KUKA KRL program: MyProgram_290().src

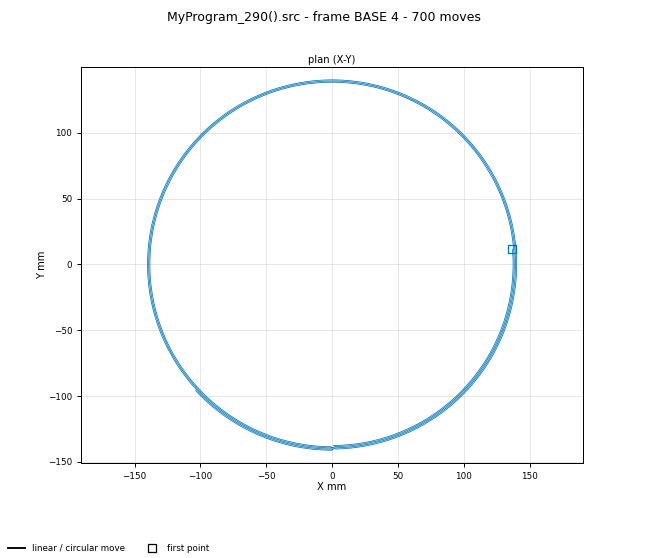
[picture p0: tool path of MyProgram_290().src in frame BASE 4, 700 of 700 moves have a stored position in this frame; points joined in program order, loops and branches not executed]
&ACCESS RVP
&REL 1
&PARAM TEMPLATE = C:\KRC\Roboter\Template\vorgabe
&PARAM EDITMASK = *
DEF MyProgram_290()
; ---- Setting reference (Base) ----
$BASE = BASE_DATA[4]

; --------------------------
; ---- Setting tool (TCP) ----
$TOOL = TOOL_DATA[3]
; --------------------------

$VEL.CP = VEL_APROX_PRINT
Startdeposition()
$VEL.CP = VEL_PRINT
LIN {X 136.961,Y 11.6597,Z 176,A 6.5071,B 7.0853,C 0.2456,E1 7.2488,E2 445.5643} C_DIS
LIN {X 137.2072,Y 8.2752,Z 176,A 5.0839,B 7.0851,C 0.2498,E1 7.2491,E2 446.9898} C_DIS
LIN {X 137.3693,Y 4.9131,Z 176,A 3.7512,B 7.0851,C 0.2525,E1 7.2492,E2 448.3148} C_DIS
LIN {X 137.4448,Y 1.8462,Z 176,A 2.5387,B 7.0849,C 0.2549,E1 7.2493,E2 449.52} C_DIS
LIN {X 137.4365,Y -2.3473,Z 176,A 0.7551,B 7.0847,C 0.2606,E1 7.2493,E2 451.3095} C_DIS
LIN {X 137.322,Y -6.1279,Z 176,A -0.7415,B 7.0847,C 0.2637,E1 7.2491,E2 452.7974} C_DIS
LIN {X 137.1485,Y -9.2287,Z 176,A -2.0117,B 7.0845,C 0.2669,E1 7.2489,E2 454.0657} C_DIS
LIN {X 136.9306,Y -12.0198,Z 176,A -3.1786,B 7.0844,C 0.2703,E1 7.2486,E2 455.2336} C_DIS
LIN {X 136.5827,Y -15.4933,Z 176,A -4.5856,B 7.0843,C 0.2736,E1 7.2482,E2 456.6358} C_DIS
LIN {X 136.1872,Y -18.6525,Z 176,A -5.8882,B 7.0841,C 0.2769,E1 7.2477,E2 457.9365} C_DIS
LIN {X 135.7668,Y -21.4897,Z 176,A -7.0624,B 7.0841,C 0.2799,E1 7.2473,E2 459.1091} C_DIS
LIN {X 135.2243,Y -24.6745,Z 176,A -8.4059,B 7.0839,C 0.2837,E1 7.2466,E2 460.4533} C_DIS
LIN {X 134.6158,Y -27.8022,Z 176,A -9.6822,B 7.0837,C 0.2865,E1 7.2459,E2 461.7243} C_DIS
LIN {X 133.8994,Y -31.0705,Z 176,A -11.0574,B 7.0837,C 0.29,E1 7.2451,E2 463.0983} C_DIS
LIN {X 133.1148,Y -34.2762,Z 176,A -12.4299,B 7.0834,C 0.2938,E1 7.2441,E2 464.4717} C_DIS
LIN {X 132.1526,Y -37.8229,Z 176,A -13.9111,B 7.0834,C 0.2972,E1 7.243,E2 465.948} C_DIS
LIN {X 131.3555,Y -40.4966,Z 176,A -15.0746,B 7.0832,C 0.3004,E1 7.2421,E2 467.1125} C_DIS
LIN {X 130.2621,Y -43.8883,Z 176,A -16.5343,B 7.083,C 0.304,E1 7.2408,E2 468.5704} C_DIS
LIN {X 129.0209,Y -47.4183,Z 176,A -18.0428,B 7.0829,C 0.3073,E1 7.2394,E2 470.074} C_DIS
LIN {X 127.9868,Y -50.1363,Z 176,A -19.2347,B 7.0828,C 0.3102,E1 7.2382,E2 471.2643} C_DIS
LIN {X 126.5088,Y -53.7624,Z 176,A -20.8363,B 7.0826,C 0.3141,E1 7.2365,E2 472.8637} C_DIS
LIN {X 125.2738,Y -56.576,Z 176,A -22.1179,B 7.0824,C 0.3175,E1 7.235,E2 474.1465} C_DIS
LIN {X 123.656,Y -60.0339,Z 176,A -23.6578,B 7.0823,C 0.3207,E1 7.2332,E2 475.6815} C_DIS
LIN {X 122.2692,Y -62.8062,Z 176,A -24.9451,B 7.0821,C 0.324,E1 7.2315,E2 476.9694} C_DIS
LIN {X 120.3748,Y -66.3676,Z 176,A -26.6709,B 7.0819,C 0.3291,E1 7.2292,E2 478.7026} C_DIS
LIN {X 118.274,Y -70.0435,Z 176,A -28.4372,B 7.0817,C 0.3336,E1 7.2268,E2 480.4708} C_DIS
LIN {X 116.0055,Y -73.7401,Z 176,A -30.1691,B 7.0815,C 0.3367,E1 7.2242,E2 482.1948} C_DIS
LIN {X 113.6894,Y -77.2622,Z 176,A -31.8872,B 7.0814,C 0.3403,E1 7.2215,E2 483.9095} C_DIS
LIN {X 111.1496,Y -80.8734,Z 176,A -33.6975,B 7.0812,C 0.3441,E1 7.2186,E2 485.7178} C_DIS
LIN {X 108.4882,Y -84.41,Z 176,A -35.4665,B 7.0811,C 0.3471,E1 7.2156,E2 487.4788} C_DIS
LIN {X 106.0889,Y -87.4067,Z 176,A -37.1314,B 7.0808,C 0.3519,E1 7.2127,E2 489.1535} C_DIS
LIN {X 103.154,Y -90.8515,Z 176,A -38.9691,B 7.0806,C 0.3553,E1 7.2093,E2 490.9868} C_DIS
LIN {X 100.4201,Y -93.8646,Z 176,A -40.5682,B 7.0806,C 0.3572,E1 7.2063,E2 492.5751} C_DIS
LIN {X 97.5463,Y -96.8473,Z 176,A -42.3208,B 7.0803,C 0.3613,E1 7.2029,E2 494.3327} C_DIS
LIN {X 94.6495,Y -99.6812,Z 176,A -43.9576,B 7.0803,C 0.3639,E1 7.1996,E2 495.9643} C_DIS
LIN {X 91.5167,Y -102.5643,Z 176,A -45.7287,B 7.08,C 0.3674,E1 7.1959,E2 497.7366} C_DIS
LIN {X 88.1549,Y -105.4678,Z 176,A -47.5543,B 7.0799,C 0.3705,E1 7.1921,E2 499.5605} C_DIS
LIN {X 84.7062,Y -108.2571,Z 176,A -49.3096,B 7.0798,C 0.3723,E1 7.1883,E2 501.3055} C_DIS
LIN {X 81.738,Y -110.5159,Z 176,A -50.8436,B 7.0796,C 0.3748,E1 7.1848,E2 502.8383} C_DIS
LIN {X 78.8688,Y -112.5814,Z 176,A -52.4099,B 7.0794,C 0.379,E1 7.1812,E2 504.4177} C_DIS
LIN {X 75.2187,Y -115.0523,Z 176,A -54.1125,B 7.0794,C 0.3797,E1 7.1773,E2 506.1046} C_DIS
LIN {X 71.7738,Y -117.2315,Z 176,A -55.8334,B 7.0792,C 0.3828,E1 7.1732,E2 507.8297} C_DIS
LIN {X 68.4893,Y -119.1809,Z 176,A -57.3647,B 7.0792,C 0.3843,E1 7.1695,E2 509.3546} C_DIS
LIN {X 65.2782,Y -120.969,Z 176,A -58.9833,B 7.0789,C 0.388,E1 7.1656,E2 510.9855} C_DIS
LIN {X 61.5873,Y -122.8897,Z 176,A -60.5947,B 7.0789,C 0.3883,E1 7.1616,E2 512.5826} C_DIS
LIN {X 58.8048,Y -124.2432,Z 176,A -61.8707,B 7.0789,C 0.3898,E1 7.1584,E2 513.8578} C_DIS
LIN {X 55.3382,Y -125.8275,Z 176,A -63.4438,B 7.0787,C 0.3916,E1 7.1544,E2 515.4301} C_DIS
LIN {X 52.6854,Y -126.9586,Z 176,A -64.6529,B 7.0787,C 0.3932,E1 7.1512,E2 516.641} C_DIS
LIN {X 49.0097,Y -128.4248,Z 176,A -66.2681,B 7.0786,C 0.3945,E1 7.1471,E2 518.2531} C_DIS
LIN {X 46.1618,Y -129.4738,Z 176,A -67.5214,B 7.0786,C 0.3957,E1 7.1438,E2 519.5057} C_DIS
LIN {X 42.9006,Y -130.591,Z 176,A -68.9539,B 7.0784,C 0.3971,E1 7.14,E2 520.9387} C_DIS
LIN {X 39.5175,Y -131.6552,Z 176,A -70.406,B 7.0784,C 0.3981,E1 7.1361,E2 522.3886} C_DIS
LIN {X 36.5593,Y -132.5059,Z 176,A -71.6852,B 7.0784,C 0.3991,E1 7.1327,E2 523.668} C_DIS
LIN {X 33.0127,Y -133.4355,Z 176,A -73.2026,B 7.0783,C 0.4002,E1 7.1286,E2 525.1851} C_DIS
LIN {X 30.3656,Y -134.0604,Z 176,A -74.339,B 7.0783,C 0.4011,E1 7.1255,E2 526.3226} C_DIS
LIN {X 26.6091,Y -134.8586,Z 176,A -75.9189,B 7.0782,C 0.4019,E1 7.1211,E2 527.9009} C_DIS
LIN {X 23.418,Y -135.4491,Z 176,A -77.2633,B 7.0782,C 0.4026,E1 7.1174,E2 529.245} C_DIS
LIN {X 20.2378,Y -135.9607,Z 176,A -78.5988,B 7.0781,C 0.4033,E1 7.1138,E2 530.5804} C_DIS
LIN {X 17.4061,Y -136.3506,Z 176,A -79.765,B 7.0781,C 0.4034,E1 7.1105,E2 531.744} C_DIS
LIN {X 14.2534,Y -136.7161,Z 176,A -81.0999,B 7.0781,C 0.4042,E1 7.1068,E2 533.0813} C_DIS
LIN {X 10.7874,Y -137.0347,Z 176,A -82.5446,B 7.0781,C 0.4046,E1 7.1028,E2 534.526} C_DIS
LIN {X 8.1562,Y -137.2145,Z 176,A -83.6805,B 7.078,C 0.4055,E1 7.0996,E2 535.6671} C_DIS
LIN {X 4.9131,Y -137.3693,Z 176,A -85.0082,B 7.078,C 0.4055,E1 7.0959,E2 536.9922} C_DIS
LIN {X 1.0091,Y -137.4517,Z 176,A -86.2503,B 7.0783,C 0.3996,E1 7.0926,E2 538.1854} C_DIS
Enddeposition()
LIN {X 1.0091,Y -137.4517,Z 176,A -86.2503,B 7.0783,C 0.3996,E1 7.0926,E2 538.1854} C_DIS
Startdeposition()
$VEL.CP = VEL_PRINT
LIN {X 2.5254,Y -138.3393,Z 176,A -85.3198,B 7.0556,C 0.3987,E1 7.0725,E2 537.2546} C_DIS
LIN {X 6.9228,Y -138.1889,Z 176,A -83.5465,B 7.0556,C 0.399,E1 7.0774,E2 535.4868} C_DIS
LIN {X 10.7421,Y -137.9461,Z 176,A -81.9791,B 7.0556,C 0.3988,E1 7.0818,E2 533.9208} C_DIS
LIN {X 13.4601,Y -137.706,Z 176,A -80.8485,B 7.0556,C 0.3984,E1 7.0849,E2 532.7896} C_DIS
LIN {X 17.2708,Y -137.2818,Z 176,A -78.452,B 7.0564,C 0.3842,E1 7.0919,E2 530.2856} C_DIS
LIN {X 23.2033,Y -136.4032,Z 176,A -76.7282,B 7.0558,C 0.3955,E1 7.0963,E2 528.6605} C_DIS
LIN {X 27.2216,Y -135.6582,Z 176,A -75.0014,B 7.0558,C 0.3938,E1 7.1011,E2 526.9282} C_DIS
LIN {X 30.8555,Y -134.8775,Z 176,A -73.2676,B 7.0561,C 0.3893,E1 7.1059,E2 525.1678} C_DIS
LIN {X 34.0474,Y -134.1073,Z 176,A -72.1782,B 7.0559,C 0.3928,E1 7.1087,E2 524.113} C_DIS
LIN {X 37.8887,Y -133.0746,Z 176,A -70.5771,B 7.0559,C 0.3921,E1 7.113,E2 522.5169} C_DIS
LIN {X 40.8202,Y -132.2037,Z 176,A -69.3143,B 7.056,C 0.391,E1 7.1164,E2 521.2536} C_DIS
LIN {X 44.7183,Y -130.9376,Z 176,A -67.5846,B 7.0561,C 0.3887,E1 7.121,E2 519.5184} C_DIS
LIN {X 48.2676,Y -129.6699,Z 176,A -66.1821,B 7.0561,C 0.3897,E1 7.1246,E2 518.1355} C_DIS
LIN {X 51.4027,Y -128.4595,Z 176,A -64.8772,B 7.0561,C 0.3897,E1 7.128,E2 516.8409} C_DIS
LIN {X 54.2024,Y -127.3051,Z 176,A -63.4709,B 7.0563,C 0.3855,E1 7.1317,E2 515.4138} C_DIS
LIN {X 56.8151,Y -126.1591,Z 176,A -62.182,B 7.0565,C 0.3821,E1 7.135,E2 514.1098} C_DIS
LIN {X 60.1001,Y -124.6281,Z 176,A -60.6977,B 7.0566,C 0.3804,E1 7.1387,E2 512.6265} C_DIS
LIN {X 63.3527,Y -123.0073,Z 176,A -59.1577,B 7.0567,C 0.3776,E1 7.1426,E2 511.0807} C_DIS
LIN {X 67.4632,Y -120.803,Z 176,A -57.3038,B 7.0568,C 0.3762,E1 7.1471,E2 509.2355} C_DIS
LIN {X 72.6683,Y -117.7453,Z 176,A -54.8126,B 7.057,C 0.3724,E1 7.1531,E2 506.7434} C_DIS
LIN {X 76.3854,Y -115.3685,Z 176,A -53.0068,B 7.0572,C 0.3697,E1 7.1573,E2 504.9387} C_DIS
LIN {X 81.0498,Y -112.1403,Z 176,A -49.8357,B 7.0581,C 0.3507,E1 7.1648,E2 501.6571} C_DIS
LIN {X 86.6426,Y -107.8779,Z 176,A -47.9887,B 7.0574,C 0.3647,E1 7.1685,E2 499.948} C_DIS
LIN {X 92.5705,Y -102.8361,Z 176,A -44.8865,B 7.0576,C 0.3606,E1 7.1751,E2 496.8588} C_DIS
LIN {X 96.6443,Y -99.0176,Z 176,A -42.3516,B 7.0581,C 0.3518,E1 7.1803,E2 494.2927} C_DIS
LIN {X 102.4902,Y -92.953,Z 176,A -39.1952,B 7.0581,C 0.3504,E1 7.1863,E2 491.1765} C_DIS
LIN {X 106.6921,Y -88.0984,Z 176,A -36.5612,B 7.0584,C 0.3449,E1 7.1911,E2 488.5434} C_DIS
LIN {X 109.9326,Y -84.0198,Z 176,A -34.3714,B 7.0587,C 0.3393,E1 7.1949,E2 486.3473} C_DIS
LIN {X 111.7517,Y -81.5857,Z 176,A -33.0115,B 7.0589,C 0.3345,E1 7.1971,E2 484.9731} C_DIS
LIN {X 114.075,Y -78.3031,Z 176,A -31.3295,B 7.0591,C 0.3301,E1 7.1998,E2 483.2873} C_DIS
LIN {X 116.3731,Y -74.8457,Z 176,A -29.6118,B 7.0593,C 0.3259,E1 7.2024,E2 481.5681} C_DIS
LIN {X 118.7096,Y -71.0817,Z 176,A -27.9699,B 7.0593,C 0.3249,E1 7.2048,E2 479.9496} C_DIS
LIN {X 120.5701,Y -67.8775,Z 176,A -26.3198,B 7.0596,C 0.3189,E1 7.2071,E2 478.2829} C_DIS
LIN {X 122.7224,Y -63.9013,Z 176,A -24.5849,B 7.0597,C 0.3166,E1 7.2094,E2 476.564} C_DIS
LIN {X 124.4953,Y -60.3781,Z 176,A -22.1195,B 7.0606,C 0.2966,E1 7.2125,E2 473.9882} C_DIS
LIN {X 127.1523,Y -54.5563,Z 176,A -20.3094,B 7.0602,C 0.3055,E1 7.2144,E2 472.2855} C_DIS
LIN {X 129.6051,Y -48.4406,Z 176,A -17.6421,B 7.0605,C 0.2993,E1 7.2171,E2 469.6237} C_DIS
LIN {X 130.7909,Y -45.1415,Z 176,A -16.2657,B 7.0605,C 0.2967,E1 7.2184,E2 468.2557} C_DIS
LIN {X 131.9779,Y -41.5469,Z 176,A -14.7467,B 7.0607,C 0.2933,E1 7.2197,E2 466.7415} C_DIS
LIN {X 133.0729,Y -37.8948,Z 176,A -13.2187,B 7.0609,C 0.2899,E1 7.2209,E2 465.2187} C_DIS
LIN {X 134.2589,Y -33.4503,Z 176,A -11.3485,B 7.0611,C 0.2852,E1 7.2222,E2 463.3511} C_DIS
LIN {X 135.0961,Y -29.8924,Z 176,A -9.8374,B 7.0612,C 0.281,E1 7.2231,E2 461.8389} C_DIS
LIN {X 136.0368,Y -25.2694,Z 176,A -7.6229,B 7.0616,C 0.2705,E1 7.2243,E2 459.5889} C_DIS
LIN {X 136.6167,Y -21.9198,Z 176,A -6.5809,B 7.0616,C 0.2734,E1 7.2248,E2 458.5929} C_DIS
LIN {X 136.9695,Y -19.5809,Z 176,A -5.5854,B 7.0616,C 0.2703,E1 7.2252,E2 457.5944} C_DIS
LIN {X 137.3908,Y -16.3656,Z 176,A -4.2291,B 7.0618,C 0.2662,E1 7.2256,E2 456.2352} C_DIS
LIN {X 138.1174,Y -8.2298,Z 176,A -1.086,B 7.062,C 0.2611,E1 7.2264,E2 453.1201} C_DIS
LIN {X 138.2614,Y -5.2795,Z 176,A 0.2729,B 7.0622,C 0.255,E1 7.2265,E2 451.7427} C_DIS
LIN {X 138.3608,Y -0.7908,Z 176,A 2.1226,B 7.0624,C 0.2498,E1 7.2265,E2 449.8927} C_DIS
LIN {X 138.3336,Y 2.8695,Z 176,A 3.5024,B 7.0624,C 0.2481,E1 7.2265,E2 448.5292} C_DIS
LIN {X 138.2205,Y 6.2935,Z 176,A 5.1475,B 7.0627,C 0.2397,E1 7.2264,E2 446.8537} C_DIS
LIN {X 137.9761,Y 10.3308,Z 176,A 6.6024,B 7.0627,C 0.2391,E1 7.2261,E2 445.4258} C_DIS
LIN {X 137.1498,Y 18.2779,Z 176,A 9.844,B 7.063,C 0.2309,E1 7.2251,E2 442.1904} C_DIS
LIN {X 136.704,Y 21.3562,Z 176,A 11.0883,B 7.0631,C 0.2281,E1 7.2246,E2 440.9507} C_DIS
LIN {X 136.1551,Y 24.6144,Z 176,A 12.4408,B 7.0632,C 0.2245,E1 7.2239,E2 439.5991} C_DIS
LIN {X 135.0836,Y 29.9503,Z 176,A 14.6215,B 7.0634,C 0.2196,E1 7.2227,E2 437.4263} C_DIS
LIN {X 134.4438,Y 32.6949,Z 176,A 15.8649,B 7.0635,C 0.2149,E1 7.2219,E2 436.1722} C_DIS
LIN {X 133.332,Y 36.9684,Z 176,A 17.6054,B 7.0636,C 0.2115,E1 7.2206,E2 434.4417} C_DIS
LIN {X 132.3059,Y 40.4861,Z 176,A 19.0601,B 7.0637,C 0.2085,E1 7.2194,E2 432.994} C_DIS
LIN {X 131.194,Y 43.9563,Z 176,A 20.5614,B 7.0638,C 0.2045,E1 7.2181,E2 431.4927} C_DIS
LIN {X 130.0878,Y 47.1295,Z 176,A 21.9276,B 7.0639,C 0.2012,E1 7.2169,E2 430.1288} C_DIS
LIN {X 128.7264,Y 50.7334,Z 176,A 23.7502,B 7.0642,C 0.1928,E1 7.215,E2 428.2762} C_DIS
LIN {X 126.8213,Y 55.322,Z 176,A 25.4906,B 7.0642,C 0.1932,E1 7.2131,E2 426.575} C_DIS
LIN {X 125.3764,Y 58.5231,Z 176,A 27.0649,B 7.0643,C 0.1872,E1 7.2113,E2 424.9847} C_DIS
LIN {X 123.8041,Y 61.7808,Z 176,A 28.3809,B 7.0643,C 0.1868,E1 7.2097,E2 423.691} C_DIS
LIN {X 122.2976,Y 64.7103,Z 176,A 29.765,B 7.0644,C 0.1829,E1 7.2079,E2 422.3036} C_DIS
LIN {X 116.9096,Y 74.0045,Z 176,A 34.0572,B 7.0646,C 0.1749,E1 7.2019,E2 418.0296} C_DIS
LIN {X 114.3482,Y 77.9047,Z 176,A 36.1172,B 7.0648,C 0.168,E1 7.1986,E2 415.9526} C_DIS
LIN {X 111.806,Y 81.5111,Z 176,A 37.9057,B 7.0648,C 0.1644,E1 7.1957,E2 414.1682} C_DIS
LIN {X 108.7844,Y 85.5012,Z 176,A 39.7845,B 7.0649,C 0.1632,E1 7.1925,E2 412.3131} C_DIS
LIN {X 106.3447,Y 88.5179,Z 176,A 41.4898,B 7.065,C 0.1579,E1 7.1895,E2 410.5948} C_DIS
LIN {X 103.8728,Y 91.4058,Z 176,A 43.0987,B 7.0651,C 0.1539,E1 7.1865,E2 408.981} C_DIS
LIN {X 100.77,Y 94.8152,Z 176,A 44.9608,B 7.0651,C 0.1507,E1 7.183,E2 407.1242} C_DIS
LIN {X 97.5573,Y 98.1176,Z 176,A 46.9196,B 7.0653,C 0.1459,E1 7.1791,E2 405.1584} C_DIS
LIN {X 94.2943,Y 101.2575,Z 176,A 48.4305,B 7.0653,C 0.1487,E1 7.1762,E2 403.693} C_DIS
LIN {X 92.1308,Y 103.2301,Z 176,A 49.8679,B 7.0653,C 0.1424,E1 7.1731,E2 402.227} C_DIS
LIN {X 88.6833,Y 106.2068,Z 176,A 51.7248,B 7.0654,C 0.1394,E1 7.1692,E2 400.3735} C_DIS
LIN {X 85.3526,Y 108.901,Z 176,A 53.4781,B 7.0654,C 0.1366,E1 7.1654,E2 398.6224} C_DIS
LIN {X 81.7479,Y 111.6325,Z 176,A 55.3312,B 7.0655,C 0.1337,E1 7.1612,E2 396.7716} C_DIS
LIN {X 74.1764,Y 116.8011,Z 176,A 59.2347,B 7.0657,C 0.1259,E1 7.1521,E2 392.8545} C_DIS
LIN {X 69.8268,Y 119.4521,Z 176,A 61.1523,B 7.0657,C 0.1261,E1 7.1476,E2 390.9609} C_DIS
LIN {X 65.895,Y 121.6656,Z 176,A 63.0289,B 7.0657,C 0.1233,E1 7.143,E2 389.0833} C_DIS
LIN {X 60.1682,Y 124.5956,Z 176,A 65.4693,B 7.0657,C 0.1237,E1 7.137,E2 386.6709} C_DIS
LIN {X 56.1062,Y 126.4762,Z 176,A 67.4503,B 7.0657,C 0.1193,E1 7.1319,E2 384.6741} C_DIS
LIN {X 51.4384,Y 128.4451,Z 176,A 69.4867,B 7.0658,C 0.118,E1 7.1267,E2 382.6455} C_DIS
LIN {X 48.0789,Y 129.7406,Z 176,A 70.9544,B 7.0658,C 0.1169,E1 7.1228,E2 381.181} C_DIS
LIN {X 45.1935,Y 130.7729,Z 176,A 72.2552,B 7.0658,C 0.1152,E1 7.1194,E2 379.8765} C_DIS
LIN {X 41.978,Y 131.8402,Z 176,A 73.6416,B 7.0658,C 0.1142,E1 7.1157,E2 378.4923} C_DIS
LIN {X 38.3573,Y 132.9398,Z 176,A 75.1467,B 7.0658,C 0.1139,E1 7.1117,E2 376.9953} C_DIS
LIN {X 34.814,Y 133.9128,Z 176,A 76.8878,B 7.066,C 0.1092,E1 7.1069,E2 375.2271} C_DIS
LIN {X 31.0115,Y 134.8419,Z 176,A 78.3311,B 7.066,C 0.111,E1 7.1031,E2 373.8064} C_DIS
LIN {X 25.4929,Y 135.9941,Z 176,A 80.5918,B 7.066,C 0.1109,E1 7.0969,E2 371.5556} C_DIS
LIN {X 22.3228,Y 136.5501,Z 176,A 82.0724,B 7.066,C 0.1078,E1 7.0928,E2 370.0569} C_DIS
LIN {X 17.0323,Y 137.3112,Z 176,A 84.0919,B 7.066,C 0.1101,E1 7.0873,E2 368.0624} C_DIS
LIN {X 12.0718,Y 137.8351,Z 176,A 86.0722,B 7.066,C 0.1108,E1 7.0818,E2 366.0935} C_DIS
LIN {X 7.3371,Y 138.168,Z 176,A 88.2612,B 7.066,C 0.1069,E1 7.0756,E2 363.8774} C_DIS
LIN {X 2.8858,Y 138.3333,Z 176,A 90.1438,B 7.066,C 0.1062,E1 7.0704,E2 361.9909} C_DIS
LIN {X -1.2214,Y 138.3576,Z 176,A 91.6876,B 7.066,C 0.1086,E1 7.0661,E2 360.4674} C_DIS
LIN {X -4.5578,Y 138.2889,Z 176,A 93.9422,B 7.0662,C 0.0953,E1 7.0595,E2 358.1041} C_DIS
LIN {X -10.7096,Y 137.9485,Z 176,A 95.5331,B 7.0659,C 0.1104,E1 7.0554,E2 356.6349} C_DIS
LIN {X -18.6513,Y 137.1008,Z 176,A 99.4322,B 7.0661,C 0.1026,E1 7.0444,E2 352.664} C_DIS
LIN {X -22.6044,Y 136.5031,Z 176,A 100.4171,B 7.0659,C 0.1134,E1 7.0419,E2 351.7636} C_DIS
LIN {X -24.5794,Y 136.1614,Z 176,A 101.5762,B 7.0659,C 0.1089,E1 7.0386,E2 350.5642} C_DIS
LIN {X -29.0231,Y 135.2838,Z 176,A 103.4719,B 7.0659,C 0.1097,E1 7.0334,E2 348.6671} C_DIS
LIN {X -32.4353,Y 134.5063,Z 176,A 104.8068,B 7.0659,C 0.1123,E1 7.0298,E2 347.3473} C_DIS
LIN {X -36.4117,Y 133.4871,Z 176,A 106.5159,B 7.0659,C 0.1134,E1 7.0252,E2 345.6383} C_DIS
LIN {X -40.6365,Y 132.2599,Z 176,A 108.3838,B 7.0659,C 0.1142,E1 7.0202,E2 343.7658} C_DIS
LIN {X -44.2376,Y 131.1004,Z 176,A 110.5174,B 7.0659,C 0.1075,E1 7.0144,E2 341.5623} C_DIS
LIN {X -48.7219,Y 129.4997,Z 176,A 111.8393,B 7.0659,C 0.1187,E1 7.0111,E2 340.3231} C_DIS
LIN {X -52.0437,Y 128.2011,Z 176,A 113.3948,B 7.0658,C 0.1192,E1 7.0071,E2 338.759} C_DIS
LIN {X -55.294,Y 126.8333,Z 176,A 114.9898,B 7.0658,C 0.1189,E1 7.0029,E2 337.1483} C_DIS
LIN {X -59.0033,Y 125.1521,Z 176,A 116.8221,B 7.0658,C 0.1189,E1 6.9982,E2 335.2991} C_DIS
LIN {X -63.5602,Y 122.9015,Z 176,A 118.7168,B 7.0658,C 0.1246,E1 6.9936,E2 333.4323} C_DIS
LIN {X -66.6076,Y 121.2769,Z 176,A 120.6249,B 7.0658,C 0.1199,E1 6.9888,E2 331.4655} C_DIS
LIN {X -70.2498,Y 119.2036,Z 176,A 121.6918,B 7.0656,C 0.1317,E1 6.9864,E2 330.4835} C_DIS
LIN {X -74.9128,Y 116.3301,Z 176,A 124.2214,B 7.0656,C 0.1315,E1 6.9803,E2 327.9232} C_DIS
LIN {X -78.1221,Y 114.1993,Z 176,A 125.9356,B 7.0656,C 0.1325,E1 6.9763,E2 326.1956} C_DIS
LIN {X -81.8457,Y 111.5606,Z 176,A 128.0751,B 7.0656,C 0.1323,E1 6.9714,E2 324.0264} C_DIS
LIN {X -84.6797,Y 109.4251,Z 176,A 129.1735,B 7.0654,C 0.1399,E1 6.9691,E2 322.9757} C_DIS
LIN {X -87.6801,Y 107.0361,Z 176,A 130.9221,B 7.0654,C 0.1406,E1 6.9653,E2 321.2085} C_DIS
LIN {X -91.1706,Y 104.0792,Z 176,A 132.9117,B 7.0654,C 0.1429,E1 6.961,E2 319.2086} C_DIS
LIN {X -94.7376,Y 100.8432,Z 176,A 134.7784,B 7.0652,C 0.1484,E1 6.9572,E2 317.3597} C_DIS
LIN {X -97.6555,Y 98.02,Z 176,A 136.5495,B 7.0652,C 0.1507,E1 6.9537,E2 315.5789} C_DIS
LIN {X -100.7775,Y 94.8073,Z 176,A 138.5403,B 7.0652,C 0.1527,E1 6.9498,E2 313.5727} C_DIS
LIN {X -104.0802,Y 91.1694,Z 176,A 140.4595,B 7.065,C 0.1586,E1 6.9463,E2 311.6699} C_DIS
LIN {X -106.5987,Y 88.2111,Z 176,A 142.1398,B 7.065,C 0.1612,E1 6.9433,E2 309.9821} C_DIS
LIN {X -109.2558,Y 84.8981,Z 176,A 143.9146,B 7.0649,C 0.165,E1 6.9402,E2 308.207} C_DIS
LIN {X -111.8062,Y 81.5108,Z 176,A 145.7743,B 7.0649,C 0.1677,E1 6.9371,E2 306.3359} C_DIS
LIN {X -114.4796,Y 77.7107,Z 176,A 147.7115,B 7.0647,C 0.1721,E1 6.934,E2 304.3989} C_DIS
LIN {X -117.2797,Y 73.4173,Z 176,A 149.575,B 7.0645,C 0.1806,E1 6.9312,E2 302.5698} C_DIS
LIN {X -118.8014,Y 70.9276,Z 176,A 151.0457,B 7.0645,C 0.1802,E1 6.9291,E2 301.0675} C_DIS
LIN {X -120.9228,Y 67.2476,Z 176,A 152.8882,B 7.0645,C 0.1836,E1 6.9265,E2 299.2162} C_DIS
LIN {X -122.8738,Y 63.6129,Z 176,A 154.7775,B 7.0644,C 0.1857,E1 6.924,E2 297.3057} C_DIS
LIN {X -125.1706,Y 58.9646,Z 176,A 156.698,B 7.0641,C 0.1941,E1 6.9218,E2 295.4157} C_DIS
LIN {X -126.2768,Y 56.5519,Z 176,A 157.9683,B 7.0641,C 0.1948,E1 6.9203,E2 294.1249} C_DIS
LIN {X -128.3795,Y 51.6012,Z 176,A 160.0918,B 7.0639,C 0.2021,E1 6.918,E2 292.0166} C_DIS
LIN {X -129.8312,Y 47.8368,Z 176,A 161.7888,B 7.0638,C 0.2063,E1 6.9163,E2 290.3179} C_DIS
LIN {X -130.6764,Y 45.4716,Z 176,A 162.8849,B 7.0638,C 0.2084,E1 6.9153,E2 289.2157} C_DIS
LIN {X -131.8419,Y 41.9728,Z 176,A 164.4104,B 7.0636,C 0.2126,E1 6.914,E2 287.6918} C_DIS
LIN {X -132.847,Y 38.6743,Z 176,A 165.8678,B 7.0636,C 0.2162,E1 6.9128,E2 286.232} C_DIS
LIN {X -133.9152,Y 34.8045,Z 176,A 167.552,B 7.0634,C 0.2205,E1 6.9116,E2 284.5467} C_DIS
LIN {X -134.6189,Y 31.9682,Z 176,A 168.7885,B 7.0633,C 0.2236,E1 6.9108,E2 283.3079} C_DIS
LIN {X -135.3494,Y 28.719,Z 176,A 170.5625,B 7.0633,C 0.2225,E1 6.9097,E2 281.4852} C_DIS
LIN {X -136.0605,Y 25.1429,Z 176,A 171.7319,B 7.063,C 0.2311,E1 6.9092,E2 280.3604} C_DIS
LIN {X -136.6305,Y 21.8312,Z 176,A 173.1103,B 7.0629,C 0.2352,E1 6.9085,E2 278.9849} C_DIS
LIN {X -136.9789,Y 19.5148,Z 176,A 174.1998,B 7.0629,C 0.2364,E1 6.9081,E2 277.8811} C_DIS
LIN {X -137.4594,Y 15.79,Z 176,A 175.9795,B 7.0629,C 0.2381,E1 6.9075,E2 276.0744} C_DIS
LIN {X -137.9915,Y 10.1209,Z 176,A 178.1946,B 7.0625,C 0.2466,E1 6.907,E2 273.8794} C_DIS
LIN {X -138.2142,Y 6.4189,Z 176,A 179.6754,B 7.0623,C 0.2517,E1 6.9067,E2 272.4069} C_DIS
LIN {X -138.316,Y 3.584,Z 176,A -179.0267,B 7.0623,C 0.2535,E1 6.9067,E2 271.0944} C_DIS
LIN {X -138.3578,Y -1.247,Z 176,A -176.89,B 7.0621,C 0.2576,E1 6.9067,E2 268.9421} C_DIS
LIN {X -138.2909,Y -4.4889,Z 176,A -175.5269,B 7.062,C 0.2612,E1 6.9067,E2 267.5776} C_DIS
LIN {X -138.0898,Y -8.6788,Z 176,A -173.859,B 7.0618,C 0.267,E1 6.907,E2 265.9199} C_DIS
LIN {X -137.761,Y -12.8878,Z 176,A -172.0353,B 7.0616,C 0.2711,E1 6.9074,E2 264.088} C_DIS
LIN {X -137.3825,Y -16.4352,Z 176,A -170.5282,B 7.0615,C 0.2749,E1 6.9079,E2 262.5782} C_DIS
LIN {X -136.9344,Y -19.8261,Z 176,A -169.1912,B 7.0613,C 0.2799,E1 6.9084,E2 261.2525} C_DIS
LIN {X -136.4284,Y -23.0524,Z 176,A -167.7791,B 7.0612,C 0.283,E1 6.9091,E2 259.8337} C_DIS
LIN {X -135.8712,Y -26.1354,Z 176,A -166.4354,B 7.061,C 0.286,E1 6.9097,E2 258.4851} C_DIS
LIN {X -135.1625,Y -29.5848,Z 176,A -164.9621,B 7.0609,C 0.2899,E1 6.9106,E2 257.011} C_DIS
LIN {X -134.4193,Y -32.7963,Z 176,A -163.5629,B 7.0607,C 0.2933,E1 6.9115,E2 255.6084} C_DIS
LIN {X -133.6143,Y -35.9345,Z 176,A -162.2415,B 7.0606,C 0.2972,E1 6.9124,E2 254.2905} C_DIS
LIN {X -132.61,Y -39.4839,Z 176,A -160.6475,B 7.0604,C 0.3006,E1 6.9137,E2 252.6891} C_DIS
LIN {X -131.703,Y -42.4075,Z 176,A -159.2818,B 7.0604,C 0.3028,E1 6.9149,E2 251.3116} C_DIS
LIN {X -130.0466,Y -47.2436,Z 176,A -157.1409,B 7.0601,C 0.3081,E1 6.9168,E2 249.169} C_DIS
LIN {X -128.3241,Y -51.7385,Z 176,A -155.0842,B 7.0599,C 0.3126,E1 6.9189,E2 247.1055} C_DIS
LIN {X -126.9679,Y -54.9828,Z 176,A -153.6414,B 7.0597,C 0.3166,E1 6.9205,E2 245.6652} C_DIS
LIN {X -125.4556,Y -58.3518,Z 176,A -152.0807,B 7.0596,C 0.3201,E1 6.9223,E2 244.1013} C_DIS
LIN {X -123.8944,Y -61.5978,Z 176,A -150.5429,B 7.0594,C 0.3233,E1 6.9242,E2 242.5585} C_DIS
LIN {X -121.2381,Y -66.6781,Z 176,A -148.2558,B 7.0591,C 0.3304,E1 6.9272,E2 240.2839} C_DIS
LIN {X -119.5646,Y -69.6342,Z 176,A -146.6081,B 7.0591,C 0.3306,E1 6.9295,E2 238.6059} C_DIS
LIN {X -117.2863,Y -73.4067,Z 176,A -144.7695,B 7.0589,C 0.3348,E1 6.9322,E2 236.7664} C_DIS
LIN {X -114.8052,Y -77.2296,Z 176,A -142.8289,B 7.0587,C 0.3385,E1 6.9352,E2 234.8198} C_DIS
LIN {X -112.2223,Y -80.9367,Z 176,A -140.9162,B 7.0585,C 0.3423,E1 6.9383,E2 232.9025} C_DIS
LIN {X -109.4986,Y -84.5849,Z 176,A -139.055,B 7.0583,C 0.3468,E1 6.9415,E2 231.0451} C_DIS
LIN {X -106.7972,Y -87.9714,Z 176,A -137.201,B 7.0582,C 0.3499,E1 6.9447,E2 229.184} C_DIS
LIN {X -103.8757,Y -91.4026,Z 176,A -135.3599,B 7.058,C 0.3541,E1 6.9481,E2 227.3467} C_DIS
LIN {X -101.1595,Y -94.3995,Z 176,A -133.6342,B 7.0578,C 0.3569,E1 6.9514,E2 225.615} C_DIS
LIN {X -98.0463,Y -97.6291,Z 176,A -131.7297,B 7.0577,C 0.3599,E1 6.9551,E2 223.7049} C_DIS
LIN {X -94.9038,Y -100.6864,Z 176,A -129.9244,B 7.0575,C 0.3635,E1 6.9587,E2 221.9014} C_DIS
LIN {X -91.9303,Y -103.4092,Z 176,A -128.1736,B 7.0574,C 0.3655,E1 6.9624,E2 220.1404} C_DIS
LIN {X -88.474,Y -106.3811,Z 176,A -126.2694,B 7.0572,C 0.3686,E1 6.9665,E2 218.2345} C_DIS
LIN {X -84.9058,Y -109.2499,Z 176,A -124.3523,B 7.0571,C 0.3715,E1 6.9707,E2 216.3149} C_DIS
LIN {X -79.3843,Y -113.3261,Z 176,A -121.7445,B 7.0567,C 0.3794,E1 6.9765,E2 213.738} C_DIS
LIN {X -75.2774,Y -116.094,Z 176,A -119.3526,B 7.0567,C 0.3776,E1 6.9822,E2 211.3019} C_DIS
LIN {X -71.1714,Y -118.6561,Z 176,A -117.4373,B 7.0565,C 0.3817,E1 6.9867,E2 209.3983} C_DIS
LIN {X -67.4222,Y -120.826,Z 176,A -115.2033,B 7.0567,C 0.3776,E1 6.9923,E2 207.1068} C_DIS
LIN {X -63.6973,Y -122.8295,Z 176,A -113.9272,B 7.0563,C 0.3867,E1 6.9953,E2 205.8927} C_DIS
LIN {X -60.8532,Y -124.2617,Z 176,A -112.6294,B 7.0562,C 0.3886,E1 6.9985,E2 204.5975} C_DIS
LIN {X -58.1944,Y -125.5284,Z 176,A -111.2678,B 7.0562,C 0.3878,E1 7.002,E2 203.2174} C_DIS
LIN {X -54.5178,Y -127.1689,Z 176,A -109.6743,B 7.056,C 0.3907,E1 7.0061,E2 201.6334} C_DIS
LIN {X -51.3166,Y -128.4942,Z 176,A -108.2341,B 7.056,C 0.392,E1 7.0098,E2 200.1922} C_DIS
LIN {X -48.4312,Y -129.6086,Z 176,A -106.899,B 7.056,C 0.3923,E1 7.0133,E2 198.8499} C_DIS
LIN {X -45.1224,Y -130.7975,Z 176,A -105.4588,B 7.0559,C 0.3938,E1 7.0171,E2 197.4115} C_DIS
LIN {X -41.3185,Y -132.0509,Z 176,A -103.8134,B 7.0558,C 0.3953,E1 7.0215,E2 195.7676} C_DIS
LIN {X -38.1212,Y -133.009,Z 176,A -102.1842,B 7.0559,C 0.3925,E1 7.0259,E2 194.1058} C_DIS
LIN {X -33.4693,Y -134.2541,Z 176,A -100.4503,B 7.0557,C 0.3977,E1 7.0305,E2 192.4054} C_DIS
LIN {X -27.2636,Y -135.6496,Z 176,A -97.8078,B 7.0556,C 0.3989,E1 7.0377,E2 189.7612} C_DIS
LIN {X -20.0589,Y -136.9011,Z 176,A -94.8682,B 7.0554,C 0.4014,E1 7.0458,E2 186.8324} C_DIS
LIN {X -17.1071,Y -137.3023,Z 176,A -93.3739,B 7.0557,C 0.3976,E1 7.05,E2 185.3036} C_DIS
LIN {X -13.139,Y -137.7368,Z 176,A -91.794,B 7.0556,C 0.399,E1 7.0544,E2 183.7325} C_DIS
LIN {X -9.5103,Y -138.036,Z 176,A -90.208,B 7.0556,C 0.3979,E1 7.0588,E2 182.1358} C_DIS
LIN {X -5.4944,Y -138.2531,Z 176,A -88.6422,B 7.0556,C 0.3995,E1 7.0632,E2 180.5822} C_DIS
LIN {X -1.3582,Y -138.3568,Z 176,A -86.8621,B 7.0556,C 0.3983,E1 7.0682,E2 178.7926} C_DIS
LIN {X -1.3582,Y -138.3568,Z 176,A -86.8621,B 7.0556,C 0.3983,E1 7.0682,E2 178.7926} C_DIS
Enddeposition()
LIN {X 1.0282,Y -139.2615,Z 176,A -86.1341,B 7.032,C 0.4064,E1 7.0469,E2 178.1377} C_DIS
Startdeposition()
$VEL.CP = VEL_PRINT
LIN {X -1.8048,Y -139.2572,Z 176,A -87.67,B 7.0317,C 0.4125,E1 7.0425,E2 179.7228} C_DIS
LIN {X -5.3362,Y -139.1656,Z 176,A -89.2451,B 7.0316,C 0.4145,E1 7.038,E2 181.3144} C_DIS
LIN {X -9.8584,Y -138.9187,Z 176,A -91.0825,B 7.0316,C 0.414,E1 7.0329,E2 183.1492} C_DIS
LIN {X -13.4981,Y -138.6122,Z 176,A -92.5369,B 7.0316,C 0.413,E1 7.0289,E2 184.598} C_DIS
LIN {X -17.4777,Y -138.1681,Z 176,A -94.2397,B 7.0316,C 0.4136,E1 7.0241,E2 186.3086} C_DIS
LIN {X -21.1208,Y -137.657,Z 176,A -95.7999,B 7.0316,C 0.4138,E1 7.0198,E2 187.8754} C_DIS
LIN {X -26.5006,Y -136.7235,Z 176,A -97.9446,B 7.0317,C 0.4114,E1 7.014,E2 190.0075} C_DIS
LIN {X -30.016,Y -135.9956,Z 176,A -99.7839,B 7.0315,C 0.4162,E1 7.0088,E2 191.8944} C_DIS
LIN {X -33.5464,Y -135.1689,Z 176,A -100.8984,B 7.0318,C 0.4096,E1 7.0059,E2 192.9603} C_DIS
LIN {X -38.51,Y -133.8389,Z 176,A -103.066,B 7.0318,C 0.4091,E1 7.0001,E2 195.1353} C_DIS
LIN {X -42.0634,Y -132.7637,Z 176,A -104.65,B 7.0318,C 0.4088,E1 6.9958,E2 196.727} C_DIS
LIN {X -45.0781,Y -131.7714,Z 176,A -106.023,B 7.0318,C 0.4088,E1 6.9921,E2 198.109} C_DIS
LIN {X -48.9972,Y -130.3637,Z 176,A -107.698,B 7.032,C 0.4067,E1 6.9878,E2 199.7792} C_DIS
LIN {X -53.2829,Y -128.6721,Z 176,A -109.5801,B 7.0321,C 0.4046,E1 6.9829,E2 201.6598} C_DIS
LIN {X -58.1856,Y -126.5303,Z 176,A -111.784,B 7.0323,C 0.4024,E1 6.9773,E2 203.8643} C_DIS
LIN {X -61.2577,Y -125.0721,Z 176,A -114.2149,B 7.0315,C 0.4156,E1 6.9709,E2 206.4281} C_DIS
LIN {X -67.84,Y -121.63,Z 176,A -116.3911,B 7.0324,C 0.3992,E1 6.9658,E2 208.4915} C_DIS
LIN {X -71.6173,Y -119.4447,Z 176,A -118.184,B 7.0326,C 0.3967,E1 6.9615,E2 210.284} C_DIS
LIN {X -76.3084,Y -116.5033,Z 176,A -120.3041,B 7.0329,C 0.3911,E1 6.9565,E2 212.3835} C_DIS
LIN {X -78.9065,Y -114.7594,Z 176,A -122.3623,B 7.0324,C 0.4,E1 6.9516,E2 214.541} C_DIS
LIN {X -83.312,Y -111.6023,Z 176,A -123.9917,B 7.0331,C 0.388,E1 6.9481,E2 216.0929} C_DIS
LIN {X -86.8271,Y -108.8899,Z 176,A -125.8757,B 7.0331,C 0.3858,E1 6.9439,E2 217.9841} C_DIS
LIN {X -90.3998,Y -105.9428,Z 176,A -127.8118,B 7.0333,C 0.3828,E1 6.9398,E2 219.9237} C_DIS
LIN {X -93.7796,Y -102.9631,Z 176,A -129.6657,B 7.0335,C 0.3794,E1 6.9359,E2 221.7773} C_DIS
LIN {X -96.9082,Y -100.0237,Z 176,A -131.4528,B 7.0337,C 0.3763,E1 6.9323,E2 223.5666} C_DIS
LIN {X -99.9534,Y -96.9808,Z 176,A -133.264,B 7.0338,C 0.3734,E1 6.9287,E2 225.3825} C_DIS
LIN {X -102.8841,Y -93.8666,Z 176,A -135.0888,B 7.034,C 0.3707,E1 6.9252,E2 227.2153} C_DIS
LIN {X -105.8795,Y -90.4743,Z 176,A -136.9817,B 7.0342,C 0.3672,E1 6.9218,E2 229.1115} C_DIS
LIN {X -108.7957,Y -86.9454,Z 176,A -138.8977,B 7.0344,C 0.3636,E1 6.9184,E2 231.031} C_DIS
LIN {X -111.6325,Y -83.2714,Z 176,A -140.8172,B 7.0346,C 0.3594,E1 6.9152,E2 232.951} C_DIS
LIN {X -114.2936,Y -79.5797,Z 176,A -142.7108,B 7.0348,C 0.3554,E1 6.9121,E2 234.8466} C_DIS
LIN {X -116.0391,Y -77.013,Z 176,A -144.0986,B 7.0348,C 0.3539,E1 6.9099,E2 236.248} C_DIS
LIN {X -118.7603,Y -72.7458,Z 176,A -146.1062,B 7.0351,C 0.348,E1 6.907,E2 238.2451} C_DIS
LIN {X -120.4491,Y -69.9142,Z 176,A -147.7874,B 7.0351,C 0.3489,E1 6.9045,E2 239.9671} C_DIS
LIN {X -122.273,Y -66.6728,Z 176,A -149.243,B 7.0353,C 0.3441,E1 6.9026,E2 241.4124} C_DIS
LIN {X -124.7317,Y -61.9477,Z 176,A -151.2536,B 7.0357,C 0.3363,E1 6.9001,E2 243.3987} C_DIS
LIN {X -126.3637,Y -58.5458,Z 176,A -152.8193,B 7.0359,C 0.3325,E1 6.8982,E2 244.9652} C_DIS
LIN {X -127.7666,Y -55.4178,Z 176,A -154.1917,B 7.0361,C 0.3283,E1 6.8967,E2 246.3319} C_DIS
LIN {X -128.8957,Y -52.7431,Z 176,A -155.7488,B 7.0361,C 0.3298,E1 6.895,E2 247.9346} C_DIS
LIN {X -130.1443,Y -49.5831,Z 176,A -156.8378,B 7.0364,C 0.3222,E1 6.8939,E2 248.9835} C_DIS
LIN {X -131.794,Y -45.013,Z 176,A -158.905,B 7.0366,C 0.3177,E1 6.892,E2 251.0581} C_DIS
LIN {X -133.0568,Y -41.1275,Z 176,A -160.4939,B 7.0368,C 0.312,E1 6.8906,E2 252.6342} C_DIS
LIN {X -133.9656,Y -38.0657,Z 176,A -162.0329,B 7.0368,C 0.3112,E1 6.8894,E2 254.2009} C_DIS
LIN {X -134.9313,Y -34.4826,Z 176,A -163.373,B 7.0371,C 0.3047,E1 6.8885,E2 255.5162} C_DIS
LIN {X -135.6827,Y -31.3979,Z 176,A -164.8734,B 7.0371,C 0.3035,E1 6.8875,E2 257.0405} C_DIS
LIN {X -136.4753,Y -27.7482,Z 176,A -166.3676,B 7.0374,C 0.2987,E1 6.8866,E2 258.5281} C_DIS
LIN {X -137.1294,Y -24.3118,Z 176,A -167.9259,B 7.0375,C 0.2961,E1 6.8858,E2 260.1004} C_DIS
LIN {X -137.8112,Y -20.0927,Z 176,A -169.696,B 7.0377,C 0.2913,E1 6.8851,E2 261.8708} C_DIS
LIN {X -138.3777,Y -15.7382,Z 176,A -171.9607,B 7.0377,C 0.2918,E1 6.8843,E2 264.192} C_DIS
LIN {X -138.7616,Y -11.864,Z 176,A -173.1802,B 7.0381,C 0.2825,E1 6.884,E2 265.3619} C_DIS
LIN {X -139.0268,Y -8.1974,Z 176,A -174.6613,B 7.0382,C 0.2778,E1 6.8837,E2 266.8378} C_DIS
LIN {X -139.2459,Y -2.4806,Z 176,A -177.6722,B 7.0382,C 0.2792,E1 6.8835,E2 269.9296} C_DIS
LIN {X -139.2501,Y 2.2305,Z 176,A -179.0861,B 7.0387,C 0.2672,E1 6.8835,E2 271.2759} C_DIS
LIN {X -139.1481,Y 5.7868,Z 176,A 179.5299,B 7.0389,C 0.262,E1 6.8837,E2 272.6486} C_DIS
LIN {X -138.9677,Y 9.1571,Z 176,A 177.7897,B 7.0389,C 0.2623,E1 6.884,E2 274.432} C_DIS
LIN {X -138.3261,Y 16.1709,Z 176,A 175.0188,B 7.0392,C 0.2525,E1 6.8847,E2 277.1843} C_DIS
LIN {X -137.8891,Y 19.5475,Z 176,A 173.5345,B 7.0393,C 0.2495,E1 6.8853,E2 278.6779} C_DIS
LIN {X -137.3771,Y 22.8693,Z 176,A 172.1726,B 7.0394,C 0.2453,E1 6.8859,E2 280.036} C_DIS
LIN {X -136.2389,Y 28.891,Z 176,A 169.6747,B 7.0397,C 0.2379,E1 6.8872,E2 282.5287} C_DIS
LIN {X -135.5376,Y 32.0219,Z 176,A 168.1953,B 7.0397,C 0.2362,E1 6.8882,E2 284.0269} C_DIS
LIN {X -134.6398,Y 35.6042,Z 176,A 166.7762,B 7.0399,C 0.2307,E1 6.8891,E2 285.432} C_DIS
LIN {X -133.8061,Y 38.6218,Z 176,A 165.3995,B 7.04,C 0.2283,E1 6.8902,E2 286.8187} C_DIS
LIN {X -132.8036,Y 41.9385,Z 176,A 163.9485,B 7.0401,C 0.2246,E1 6.8914,E2 288.2716} C_DIS
LIN {X -131.7266,Y 45.2074,Z 176,A 162.4369,B 7.0402,C 0.222,E1 6.8928,E2 289.7938} C_DIS
LIN {X -130.5089,Y 48.6096,Z 176,A 161.001,B 7.0404,C 0.2173,E1 6.8941,E2 291.222} C_DIS
LIN {X -129.1933,Y 52.0048,Z 176,A 159.5321,B 7.0404,C 0.2129,E1 6.8956,E2 292.6857} C_DIS
LIN {X -128.0452,Y 54.7732,Z 176,A 158.143,B 7.0405,C 0.2116,E1 6.8971,E2 294.0932} C_DIS
LIN {X -126.7961,Y 57.609,Z 176,A 156.9031,B 7.0406,C 0.2078,E1 6.8986,E2 295.3276} C_DIS
LIN {X -124.4464,Y 62.5221,Z 176,A 154.503,B 7.0408,C 0.204,E1 6.9015,E2 297.7456} C_DIS
LIN {X -122.4699,Y 66.3119,Z 176,A 152.5739,B 7.0408,C 0.2017,E1 6.9041,E2 299.6943} C_DIS
LIN {X -119.8468,Y 70.9427,Z 176,A 150.6235,B 7.0411,C 0.1932,E1 6.9068,E2 301.6129} C_DIS
LIN {X -116.6787,Y 76.0401,Z 176,A 147.9872,B 7.0411,C 0.1893,E1 6.9107,E2 304.2676} C_DIS
LIN {X -114.1181,Y 79.8319,Z 176,A 146.0805,B 7.0413,C 0.1851,E1 6.9137,E2 306.1756} C_DIS
LIN {X -112.1923,Y 82.5157,Z 176,A 144.6615,B 7.0413,C 0.1827,E1 6.9161,E2 307.6007} C_DIS
LIN {X -109.2987,Y 86.3126,Z 176,A 142.7564,B 7.0415,C 0.1775,E1 6.9193,E2 309.4968} C_DIS
LIN {X -106.5894,Y 89.6363,Z 176,A 141.0786,B 7.0415,C 0.1725,E1 6.9223,E2 311.1621} C_DIS
LIN {X -103.6527,Y 93.0166,Z 176,A 138.6404,B 7.0415,C 0.1762,E1 6.9269,E2 313.6726} C_DIS
LIN {X -100.709,Y 96.1959,Z 176,A 137.2286,B 7.0417,C 0.1677,E1 6.9295,E2 315.0369} C_DIS
LIN {X -97.4516,Y 99.4944,Z 176,A 134.8465,B 7.0417,C 0.17,E1 6.9344,E2 317.4759} C_DIS
LIN {X -94.1116,Y 102.6596,Z 176,A 133.0145,B 7.0417,C 0.1655,E1 6.9381,E2 319.2988} C_DIS
LIN {X -91.0326,Y 105.3994,Z 176,A 131.6413,B 7.0419,C 0.158,E1 6.9409,E2 320.6306} C_DIS
LIN {X -87.5822,Y 108.2836,Z 176,A 130.0045,B 7.0421,C 0.1518,E1 6.9444,E2 322.2393} C_DIS
LIN {X -81.7382,Y 112.76,Z 176,A 126.7106,B 7.0421,C 0.1501,E1 6.9518,E2 325.5637} C_DIS
LIN {X -77.9906,Y 115.3838,Z 176,A 124.821,B 7.0421,C 0.1472,E1 6.9561,E2 327.4526} C_DIS
LIN {X -74.222,Y 117.8434,Z 176,A 122.9975,B 7.0422,C 0.1439,E1 6.9604,E2 329.2712} C_DIS
LIN {X -71.0115,Y 119.8054,Z 176,A 120.9654,B 7.0422,C 0.1482,E1 6.9654,E2 331.3617} C_DIS
LIN {X -67.2023,Y 121.9831,Z 176,A 119.5122,B 7.0422,C 0.1409,E1 6.9689,E2 332.7702} C_DIS
LIN {X -63.4769,Y 123.9604,Z 176,A 117.9998,B 7.0424,C 0.1355,E1 6.9725,E2 334.2535} C_DIS
LIN {X -61.526,Y 124.9397,Z 176,A 116.3928,B 7.0422,C 0.1442,E1 6.9768,E2 335.9474} C_DIS
LIN {X -57.111,Y 127.0189,Z 176,A 114.9361,B 7.0424,C 0.1341,E1 6.9803,E2 337.3347} C_DIS
LIN {X -53.8439,Y 128.4378,Z 176,A 113.7157,B 7.0425,C 0.129,E1 6.9834,E2 338.5236} C_DIS
LIN {X -50.1258,Y 129.9344,Z 176,A 111.477,B 7.0425,C 0.1356,E1 6.9894,E2 340.8342} C_DIS
LIN {X -46.799,Y 131.1697,Z 176,A 110.2015,B 7.0425,C 0.1316,E1 6.9927,E2 342.0859} C_DIS
LIN {X -42.5261,Y 132.6159,Z 176,A 108.5718,B 7.0425,C 0.1267,E1 6.9969,E2 343.6863} C_DIS
LIN {X -39.2488,Y 133.6225,Z 176,A 107.1903,B 7.0425,C 0.1251,E1 7.0006,E2 345.0633} C_DIS
LIN {X -37.1145,Y 134.2316,Z 176,A 106.1108,B 7.0425,C 0.1268,E1 7.0035,E2 346.1628} C_DIS
LIN {X -33.017,Y 135.2978,Z 176,A 104.5141,B 7.0426,C 0.1235,E1 7.0078,E2 347.7404} C_DIS
LIN {X -30.1719,Y 135.9623,Z 176,A 103.0464,B 7.0426,C 0.1266,E1 7.0119,E2 349.2404} C_DIS
LIN {X -26.1747,Y 136.7858,Z 176,A 101.4429,B 7.0426,C 0.1246,E1 7.0163,E2 350.8334} C_DIS
LIN {X -19.0491,Y 137.9604,Z 176,A 98.3982,B 7.0426,C 0.1244,E1 7.0247,E2 353.8856} C_DIS
LIN {X -10.9424,Y 138.8395,Z 176,A 95.1733,B 7.0426,C 0.1215,E1 7.0336,E2 357.0927} C_DIS
LIN {X -4.9683,Y 139.18,Z 176,A 92.698,B 7.0426,C 0.1214,E1 7.0405,E2 359.5685} C_DIS
LIN {X -0.9708,Y 139.2647,Z 176,A 91.0788,B 7.0426,C 0.1209,E1 7.045,E2 361.1838} C_DIS
LIN {X 2.163,Y 139.2512,Z 176,A 89.6745,B 7.0426,C 0.1227,E1 7.049,E2 362.6017} C_DIS
LIN {X 6.4631,Y 139.1188,Z 176,A 88.0359,B 7.0426,C 0.1209,E1 7.0535,E2 364.2234} C_DIS
LIN {X 9.9587,Y 138.9114,Z 176,A 86.4649,B 7.0426,C 0.1232,E1 7.0579,E2 365.81} C_DIS
LIN {X 14.4172,Y 138.5204,Z 176,A 84.8394,B 7.0426,C 0.1203,E1 7.0624,E2 367.408} C_DIS
LIN {X 18.0226,Y 138.0967,Z 176,A 82.521,B 7.0424,C 0.1338,E1 7.0691,E2 369.8278} C_DIS
LIN {X 23.5428,Y 137.2648,Z 176,A 80.9343,B 7.0426,C 0.1237,E1 7.0732,E2 371.3263} C_DIS
LIN {X 29.9276,Y 136.0151,Z 176,A 78.2582,B 7.0426,C 0.1253,E1 7.0805,E2 374.0016} C_DIS
LIN {X 35.1761,Y 134.7539,Z 176,A 75.9704,B 7.0426,C 0.1279,E1 7.0867,E2 376.2972} C_DIS
LIN {X 39.0749,Y 133.6735,Z 176,A 74.4471,B 7.0426,C 0.1269,E1 7.0908,E2 377.8026} C_DIS
LIN {X 41.9127,Y 132.8119,Z 176,A 73.1126,B 7.0426,C 0.1298,E1 7.0944,E2 379.1511} C_DIS
LIN {X 45.0116,Y 131.7945,Z 176,A 71.7632,B 7.0425,C 0.1312,E1 7.098,E2 380.5012} C_DIS
LIN {X 48.2387,Y 130.6479,Z 176,A 70.3409,B 7.0425,C 0.1328,E1 7.1017,E2 381.925} C_DIS
LIN {X 52.3462,Y 129.0557,Z 176,A 68.2656,B 7.0423,C 0.139,E1 7.1072,E2 384.0327} C_DIS
LIN {X 56.0176,Y 127.5072,Z 176,A 67.022,B 7.0424,C 0.1344,E1 7.1102,E2 385.2272} C_DIS
LIN {X 64.963,Y 123.1878,Z 176,A 63.0137,B 7.0424,C 0.1383,E1 7.1203,E2 389.2257} C_DIS
LIN {X 68.5971,Y 121.2046,Z 176,A 61.1636,B 7.0423,C 0.1431,E1 7.1248,E2 391.0942} C_DIS
LIN {X 72.5198,Y 118.8989,Z 176,A 59.3148,B 7.0423,C 0.1455,E1 7.1292,E2 392.9402} C_DIS
LIN {X 75.8664,Y 116.7914,Z 176,A 57.595,B 7.0421,C 0.1496,E1 7.1333,E2 394.6716} C_DIS
LIN {X 80.5996,Y 113.5773,Z 176,A 55.3834,B 7.0421,C 0.151,E1 7.1383,E2 396.8658} C_DIS
LIN {X 84.2268,Y 110.9142,Z 176,A 53.5447,B 7.0421,C 0.154,E1 7.1424,E2 398.7031} C_DIS
LIN {X 87.6705,Y 108.2124,Z 176,A 51.7781,B 7.042,C 0.1566,E1 7.1463,E2 400.4658} C_DIS
LIN {X 91.1963,Y 105.2584,Z 176,A 49.9215,B 7.042,C 0.1595,E1 7.1502,E2 402.3183} C_DIS
LIN {X 93.7506,Y 102.9894,Z 176,A 48.7422,B 7.042,C 0.1582,E1 7.1526,E2 403.4694} C_DIS
LIN {X 98.0285,Y 98.9262,Z 176,A 46.1377,B 7.0418,C 0.1661,E1 7.1579,E2 406.0969} C_DIS
LIN {X 101.1464,Y 95.7361,Z 176,A 44.325,B 7.0417,C 0.1695,E1 7.1614,E2 407.9073} C_DIS
LIN {X 104.2899,Y 92.3015,Z 176,A 42.4783,B 7.0417,C 0.1724,E1 7.1649,E2 409.7459} C_DIS
LIN {X 106.9686,Y 89.1842,Z 176,A 40.8665,B 7.0415,C 0.1747,E1 7.1678,E2 411.3484} C_DIS
LIN {X 111.0288,Y 84.075,Z 176,A 38.1418,B 7.0414,C 0.1814,E1 7.1725,E2 414.0791} C_DIS
LIN {X 113.6383,Y 80.5132,Z 176,A 36.3381,B 7.0413,C 0.1854,E1 7.1754,E2 415.882} C_DIS
LIN {X 115.7752,Y 77.4083,Z 176,A 34.8492,B 7.0413,C 0.188,E1 7.1777,E2 417.3638} C_DIS
LIN {X 118.188,Y 73.672,Z 176,A 32.6695,B 7.0409,C 0.1987,E1 7.181,E2 419.5883} C_DIS
LIN {X 120.3976,Y 70.0017,Z 176,A 31.0881,B 7.0409,C 0.1998,E1 7.1832,E2 421.1478} C_DIS
LIN {X 122.1379,Y 66.9205,Z 176,A 29.8628,B 7.0409,C 0.1992,E1 7.1848,E2 422.3449} C_DIS
LIN {X 124.0305,Y 63.3391,Z 176,A 28.3869,B 7.0409,C 0.2,E1 7.1867,E2 423.7974} C_DIS
LIN {X 126.6547,Y 57.9166,Z 176,A 25.8952,B 7.0407,C 0.2066,E1 7.1897,E2 426.2923} C_DIS
LIN {X 129.4916,Y 51.2647,Z 176,A 22.961,B 7.0405,C 0.2137,E1 7.1929,E2 429.2232} C_DIS
LIN {X 130.9027,Y 47.5395,Z 176,A 21.3545,B 7.0404,C 0.2175,E1 7.1944,E2 430.8265} C_DIS
LIN {X 131.882,Y 44.7572,Z 176,A 20.0704,B 7.0402,C 0.2221,E1 7.1956,E2 432.1205} C_DIS
LIN {X 133.1644,Y 40.776,Z 176,A 18.4771,B 7.0402,C 0.2244,E1 7.1969,E2 433.6987} C_DIS
LIN {X 134.1605,Y 37.3688,Z 176,A 17.0797,B 7.0401,C 0.2273,E1 7.198,E2 435.089} C_DIS
LIN {X 135.095,Y 33.8377,Z 176,A 15.5836,B 7.0399,C 0.2313,E1 7.199,E2 436.5854} C_DIS
LIN {X 136.3833,Y 28.2001,Z 176,A 13.0763,B 7.0396,C 0.2404,E1 7.2006,E2 439.1107} C_DIS
LIN {X 137.0615,Y 24.6911,Z 176,A 10.8548,B 7.039,C 0.2585,E1 7.2017,E2 441.4282} C_DIS
LIN {X 138.1498,Y 17.6175,Z 176,A 8.4372,B 7.039,C 0.2571,E1 7.2025,E2 443.7818} C_DIS
LIN {X 138.6424,Y 13.1836,Z 176,A 7.1875,B 7.0392,C 0.2514,E1 7.2029,E2 444.9583} C_DIS
LIN {X 138.8799,Y 10.3909,Z 176,A 5.9313,B 7.039,C 0.2566,E1 7.2032,E2 446.2286} C_DIS
LIN {X 139.1476,Y 5.7998,Z 176,A 4.1074,B 7.0389,C 0.2608,E1 7.2034,E2 448.0454} C_DIS
LIN {X 139.2544,Y 1.9674,Z 176,A 2.5849,B 7.0388,C 0.2642,E1 7.2035,E2 449.5622} C_DIS
LIN {X 139.2593,Y -1.6743,Z 176,A 1.0885,B 7.0386,C 0.2685,E1 7.2035,E2 451.0597} C_DIS
LIN {X 139.1507,Y -5.7198,Z 176,A -0.5354,B 7.0385,C 0.2725,E1 7.2033,E2 452.6796} C_DIS
LIN {X 138.9907,Y -8.7842,Z 176,A -1.7695,B 7.0383,C 0.2756,E1 7.2031,E2 453.9113} C_DIS
LIN {X 138.5254,Y -14.3702,Z 176,A -4.0333,B 7.0381,C 0.2815,E1 7.2026,E2 456.1717} C_DIS
LIN {X 138.1018,Y -17.9834,Z 176,A -5.4778,B 7.038,C 0.2847,E1 7.2021,E2 457.6107} C_DIS
LIN {X 137.2465,Y -23.6525,Z 176,A -7.8205,B 7.0377,C 0.2912,E1 7.201,E2 459.9536} C_DIS
LIN {X 136.5502,Y -27.3801,Z 176,A -9.3585,B 7.0375,C 0.2952,E1 7.2002,E2 461.4902} C_DIS
LIN {X 135.7179,Y -31.2435,Z 176,A -10.9076,B 7.0375,C 0.2983,E1 7.1993,E2 463.0309} C_DIS
LIN {X 134.4267,Y -36.4034,Z 176,A -13.4271,B 7.0369,C 0.3107,E1 7.1975,E2 465.595} C_DIS
LIN {X 133.3425,Y -40.194,Z 176,A -14.739,B 7.0369,C 0.3093,E1 7.1965,E2 466.8685} C_DIS
LIN {X 132.3366,Y -43.3918,Z 176,A -16.0328,B 7.0369,C 0.3116,E1 7.1954,E2 468.1526} C_DIS
LIN {X 131.1236,Y -46.9269,Z 176,A -17.2929,B 7.0369,C 0.3105,E1 7.1942,E2 469.3783} C_DIS
LIN {X 130.102,Y -49.6926,Z 176,A -18.8446,B 7.0365,C 0.3202,E1 7.1927,E2 470.9751} C_DIS
LIN {X 128.5627,Y -53.545,Z 176,A -20.2572,B 7.0365,C 0.3193,E1 7.1912,E2 472.3512} C_DIS
LIN {X 125.492,Y -60.3929,Z 176,A -23.3658,B 7.0361,C 0.3279,E1 7.1876,E2 475.4656} C_DIS
LIN {X 123.3425,Y -64.6685,Z 176,A -25.2959,B 7.0359,C 0.3323,E1 7.1852,E2 477.3926} C_DIS
LIN {X 121.2703,Y -68.4802,Z 176,A -27.1356,B 7.0356,C 0.3379,E1 7.1827,E2 479.2412} C_DIS
LIN {X 119.47,Y -71.5749,Z 176,A -28.8714,B 7.0352,C 0.3464,E1 7.1802,E2 481.0124} C_DIS
LIN {X 117.4933,Y -74.7757,Z 176,A -30.1565,B 7.0352,C 0.3454,E1 7.1783,E2 482.2651} C_DIS
LIN {X 114.8931,Y -78.7117,Z 176,A -32.0091,B 7.0352,C 0.3485,E1 7.1754,E2 484.1082} C_DIS
LIN {X 112.0584,Y -82.698,Z 176,A -33.7247,B 7.0352,C 0.3478,E1 7.1727,E2 485.7871} C_DIS
LIN {X 108.1774,Y -87.7138,Z 176,A -36.589,B 7.0346,C 0.3586,E1 7.1677,E2 488.6871} C_DIS
LIN {X 106.2463,Y -90.0428,Z 176,A -37.981,B 7.0343,C 0.3641,E1 7.1652,E2 490.0995} C_DIS
LIN {X 104.0889,Y -92.5289,Z 176,A -39.148,B 7.0343,C 0.3637,E1 7.163,E2 491.2435} C_DIS
LIN {X 99.2706,Y -97.6798,Z 176,A -41.9981,B 7.0341,C 0.369,E1 7.1576,E2 494.0896} C_DIS
LIN {X 96.1434,Y -100.7591,Z 176,A -43.7585,B 7.0339,C 0.3719,E1 7.154,E2 495.8458} C_DIS
LIN {X 92.6015,Y -104.0239,Z 176,A -46.2137,B 7.0333,C 0.3844,E1 7.1488,E2 498.3642} C_DIS
LIN {X 88.8271,Y -107.2646,Z 176,A -47.716,B 7.0336,C 0.3786,E1 7.1457,E2 499.7978} C_DIS
LIN {X 85.6329,Y -109.8322,Z 176,A -49.593,B 7.0332,C 0.3852,E1 7.1416,E2 501.7012} C_DIS
LIN {X 83.0413,Y -111.8039,Z 176,A -50.6497,B 7.0334,C 0.3825,E1 7.1393,E2 502.7222} C_DIS
LIN {X 77.8501,Y -115.4789,Z 176,A -53.3247,B 7.0331,C 0.3881,E1 7.1331,E2 505.4072} C_DIS
LIN {X 75.16,Y -117.2473,Z 176,A -55.4729,B 7.0321,C 0.4048,E1 7.1278,E2 507.663} C_DIS
LIN {X 69.1823,Y -120.871,Z 176,A -57.459,B 7.0327,C 0.3937,E1 7.1233,E2 509.5365} C_DIS
LIN {X 65.357,Y -122.9809,Z 176,A -59.2436,B 7.0327,C 0.3961,E1 7.1189,E2 511.3209} C_DIS
LIN {X 62.7732,Y -124.3186,Z 176,A -60.4507,B 7.0325,C 0.3979,E1 7.1159,E2 512.5303} C_DIS
LIN {X 58.7679,Y -126.261,Z 176,A -61.9625,B 7.0327,C 0.3948,E1 7.1122,E2 514.0018} C_DIS
LIN {X 56.834,Y -127.1428,Z 176,A -63.3683,B 7.0321,C 0.4051,E1 7.1084,E2 515.4776} C_DIS
LIN {X 53.4273,Y -128.6118,Z 176,A -64.5592,B 7.0323,C 0.4012,E1 7.1055,E2 516.626} C_DIS
LIN {X 49.7175,Y -130.0931,Z 176,A -66.2475,B 7.0322,C 0.4039,E1 7.1011,E2 518.3215} C_DIS
LIN {X 44.7983,Y -131.8683,Z 176,A -68.4495,B 7.032,C 0.4071,E1 7.0952,E2 520.5316} C_DIS
LIN {X 40.9523,Y -133.1104,Z 176,A -69.9766,B 7.032,C 0.4064,E1 7.0912,E2 522.0421} C_DIS
LIN {X 37.4973,Y -134.1245,Z 176,A -71.4123,B 7.032,C 0.4069,E1 7.0874,E2 523.4729} C_DIS
LIN {X 29.6548,Y -136.074,Z 176,A -74.5978,B 7.032,C 0.4073,E1 7.0788,E2 526.6424} C_DIS
LIN {X 23.7004,Y -137.2385,Z 176,A -77.6508,B 7.0313,C 0.4181,E1 7.0702,E2 529.7696} C_DIS
LIN {X 19.719,Y -137.8646,Z 176,A -78.9763,B 7.0316,C 0.4135,E1 7.0666,E2 531.0529} C_DIS
LIN {X 15.5632,Y -138.397,Z 176,A -80.5792,B 7.0316,C 0.4123,E1 7.0622,E2 532.641} C_DIS
LIN {X 12.2142,Y -138.732,Z 176,A -82.0359,B 7.0316,C 0.414,E1 7.0581,E2 534.1079} C_DIS
LIN {X 8.3235,Y -139.0191,Z 176,A -83.5565,B 7.0316,C 0.4132,E1 7.0539,E2 535.6183} C_DIS
LIN {X 4.1632,Y -139.206,Z 176,A -85.3088,B 7.0316,C 0.4142,E1 7.049,E2 537.3766} C_DIS
LIN {X 1.0282,Y -139.2615,Z 176,A -86.1307,B 7.032,C 0.4068,E1 7.0469,E2 538.1377} C_DIS
Enddeposition()
LIN {X 1.0282,Y -139.2615,Z 176,A -86.1307,B 7.032,C 0.4068,E1 7.0469,E2 538.1377} C_DIS
Startdeposition()
$VEL.CP = VEL_PRINT
LIN {X 2.6164,Y -140.1495,Z 176,A -85.2321,B 6.9499,C 0.4068,E1 6.9673,E2 537.2625} C_DIS
LIN {X 6.2713,Y -140.0353,Z 176,A -83.5935,B 6.95,C 0.404,E1 6.972,E2 535.604} C_DIS
LIN {X 10.3448,Y -139.7913,Z 176,A -82.0867,B 6.95,C 0.4061,E1 6.9761,E2 534.1177} C_DIS
LIN {X 13.4231,Y -139.5293,Z 176,A -80.7531,B 6.95,C 0.4045,E1 6.9798,E2 532.774} C_DIS
LIN {X 16.7585,Y -139.1681,Z 176,A -79.4685,B 6.95,C 0.4053,E1 6.9834,E2 531.5002} C_DIS
LIN {X 22.4788,Y -138.3605,Z 176,A -77.1006,B 6.95,C 0.404,E1 6.9899,E2 529.1301} C_DIS
LIN {X 26.3052,Y -137.683,Z 176,A -75.4987,B 6.9501,C 0.4027,E1 6.9943,E2 527.5254} C_DIS
LIN {X 29.9782,Y -136.9307,Z 176,A -73.8859,B 6.9503,C 0.4003,E1 6.9988,E2 525.901} C_DIS
LIN {X 36.7559,Y -135.27,Z 176,A -71.2604,B 6.9502,C 0.4018,E1 7.0058,E2 523.3038} C_DIS
LIN {X 41.0843,Y -134.0172,Z 176,A -69.3311,B 6.9503,C 0.3986,E1 7.011,E2 521.3616} C_DIS
LIN {X 46.9259,Y -132.0867,Z 176,A -66.8936,B 6.9504,C 0.3974,E1 7.0175,E2 518.9327} C_DIS
LIN {X 49.8636,Y -131.0064,Z 176,A -65.5736,B 6.9505,C 0.3952,E1 7.0209,E2 517.6064} C_DIS
LIN {X 52.6484,Y -129.9104,Z 176,A -64.3035,B 6.9507,C 0.393,E1 7.0242,E2 516.3291} C_DIS
LIN {X 59.355,Y -126.9874,Z 176,A -61.2821,B 6.9509,C 0.3886,E1 7.032,E2 513.3013} C_DIS
LIN {X 63.3661,Y -125.0331,Z 176,A -59.7854,B 6.9507,C 0.3919,E1 7.0356,E2 511.8467} C_DIS
LIN {X 66.4523,Y -123.4226,Z 176,A -58.0774,B 6.9511,C 0.3848,E1 7.0399,E2 510.0998} C_DIS
LIN {X 70.6413,Y -121.074,Z 176,A -55.1022,B 6.9523,C 0.3637,E1 7.0474,E2 506.987} C_DIS
LIN {X 77.4408,Y -116.8424,Z 176,A -53.1531,B 6.9513,C 0.3821,E1 7.0516,E2 505.2128} C_DIS
LIN {X 82.0281,Y -113.6684,Z 176,A -50.6015,B 6.9517,C 0.3733,E1 7.0575,E2 502.6232} C_DIS
LIN {X 84.8133,Y -111.6061,Z 176,A -49.276,B 6.9517,C 0.3724,E1 7.0604,E2 501.3085} C_DIS
LIN {X 88.1259,Y -109.0086,Z 176,A -47.5302,B 6.952,C 0.3687,E1 7.0643,E2 499.5579} C_DIS
LIN {X 92.6323,Y -105.2063,Z 176,A -45.1004,B 6.9523,C 0.3636,E1 7.0694,E2 497.1232} C_DIS
LIN {X 95.8109,Y -102.3203,Z 176,A -43.4528,B 6.9523,C 0.362,E1 7.0728,E2 495.4884} C_DIS
LIN {X 98.8013,Y -99.4351,Z 176,A -41.8011,B 6.9525,C 0.3593,E1 7.076,E2 493.8413} C_DIS
LIN {X 102.6409,Y -95.4667,Z 176,A -39.3093,B 6.9529,C 0.3501,E1 7.0809,E2 491.3161} C_DIS
LIN {X 105.0277,Y -92.8344,Z 176,A -38.1723,B 6.9529,C 0.3528,E1 7.0829,E2 490.2198} C_DIS
LIN {X 107.7336,Y -89.6807,Z 176,A -36.4131,B 6.9531,C 0.3478,E1 7.0861,E2 488.4509} C_DIS
LIN {X 112.0587,Y -84.2138,Z 176,A -33.7002,B 6.9533,C 0.3437,E1 7.0908,E2 485.7535} C_DIS
LIN {X 115.5402,Y -79.3695,Z 176,A -31.4931,B 6.9533,C 0.3422,E1 7.0943,E2 483.5747} C_DIS
LIN {X 117.0885,Y -77.067,Z 176,A -30.0516,B 6.9537,C 0.3337,E1 7.0966,E2 482.0914} C_DIS
LIN {X 120.2304,Y -72.0682,Z 176,A -28.0313,B 6.9537,C 0.335,E1 7.0995,E2 480.1208} C_DIS
LIN {X 121.7001,Y -69.5567,Z 176,A -26.602,B 6.954,C 0.3275,E1 7.1015,E2 478.6587} C_DIS
LIN {X 123.8258,Y -65.6963,Z 176,A -24.7313,B 6.9543,C 0.3216,E1 7.104,E2 476.777} C_DIS
LIN {X 126.1197,Y -61.1801,Z 176,A -22.8905,B 6.9543,C 0.3205,E1 7.1062,E2 474.9647} C_DIS
LIN {X 127.86,Y -57.4487,Z 176,A -21.3498,B 6.9544,C 0.3187,E1 7.108,E2 473.441} C_DIS
LIN {X 129.5219,Y -53.5982,Z 176,A -19.4419,B 6.9548,C 0.3105,E1 7.1101,E2 471.506} C_DIS
LIN {X 131.0411,Y -49.7709,Z 176,A -17.6977,B 6.9551,C 0.3048,E1 7.1119,E2 469.7522} C_DIS
LIN {X 132.6171,Y -45.4038,Z 176,A -15.9115,B 6.9552,C 0.3017,E1 7.1135,E2 467.9789} C_DIS
LIN {X 133.9755,Y -41.2205,Z 176,A -14.1579,B 6.9554,C 0.2976,E1 7.115,E2 466.2294} C_DIS
LIN {X 135.654,Y -35.3161,Z 176,A -11.6507,B 6.9557,C 0.2906,E1 7.1169,E2 463.7203} C_DIS
LIN {X 136.7237,Y -30.9078,Z 176,A -9.9835,B 6.9557,C 0.2889,E1 7.1179,E2 462.0759} C_DIS
LIN {X 137.9241,Y -25.0121,Z 176,A -7.5234,B 6.956,C 0.282,E1 7.1192,E2 459.6134} C_DIS
LIN {X 138.6077,Y -20.8998,Z 176,A -5.9101,B 6.9562,C 0.2788,E1 7.1199,E2 458.0106} C_DIS
LIN {X 139.1343,Y -17.0421,Z 176,A -4.2909,B 6.9564,C 0.2738,E1 7.1205,E2 456.3863} C_DIS
LIN {X 139.5655,Y -13.0461,Z 176,A -2.4184,B 6.9567,C 0.2647,E1 7.121,E2 454.4821} C_DIS
LIN {X 139.864,Y -9.3385,Z 176,A -1.3119,B 6.9566,C 0.2682,E1 7.1212,E2 453.4287} C_DIS
LIN {X 140.08,Y -5.1323,Z 176,A 0.4105,B 6.9568,C 0.2632,E1 7.1214,E2 451.7047} C_DIS
LIN {X 140.168,Y -1.4275,Z 176,A 1.8867,B 6.9568,C 0.2596,E1 7.1215,E2 450.2322} C_DIS
LIN {X 140.1526,Y 2.4267,Z 176,A 3.4791,B 6.9571,C 0.2548,E1 7.1215,E2 448.6362} C_DIS
LIN {X 140.0203,Y 6.5703,Z 176,A 4.9746,B 6.9571,C 0.2537,E1 7.1213,E2 447.1654} C_DIS
LIN {X 139.7842,Y 10.4423,Z 176,A 6.6176,B 6.9573,C 0.2481,E1 7.121,E2 445.5136} C_DIS
LIN {X 139.4736,Y 14.0035,Z 176,A 8.332,B 6.9576,C 0.2391,E1 7.1206,E2 443.765} C_DIS
LIN {X 138.5242,Y 21.4391,Z 176,A 10.7962,B 6.9576,C 0.2417,E1 7.1197,E2 441.3766} C_DIS
LIN {X 138.0552,Y 24.2795,Z 176,A 12.2948,B 6.9579,C 0.2323,E1 7.119,E2 439.8354} C_DIS
LIN {X 137.3101,Y 28.1877,Z 176,A 13.8706,B 6.9579,C 0.2287,E1 7.1181,E2 438.2649} C_DIS
LIN {X 136.491,Y 31.9259,Z 176,A 15.4564,B 6.9581,C 0.2239,E1 7.1171,E2 436.6753} C_DIS
LIN {X 135.3772,Y 36.3539,Z 176,A 17.2125,B 6.9582,C 0.2208,E1 7.1159,E2 434.9322} C_DIS
LIN {X 134.3222,Y 40.0825,Z 176,A 18.7552,B 6.9583,C 0.2173,E1 7.1147,E2 433.3939} C_DIS
LIN {X 133.4854,Y 42.7806,Z 176,A 19.9151,B 6.9584,C 0.214,E1 7.1137,E2 432.2324} C_DIS
LIN {X 132.2526,Y 46.4553,Z 176,A 21.4362,B 6.9585,C 0.2109,E1 7.1123,E2 430.7185} C_DIS
LIN {X 131.1236,Y 49.5508,Z 176,A 22.8137,B 6.9587,C 0.2067,E1 7.111,E2 429.3362} C_DIS
LIN {X 128.0776,Y 56.9623,Z 176,A 25.9759,B 6.9588,C 0.2002,E1 7.1076,E2 426.1868} C_DIS
LIN {X 125.5779,Y 62.2796,Z 176,A 28.3618,B 6.959,C 0.1943,E1 7.1047,E2 423.8017} C_DIS
LIN {X 123.7388,Y 65.8619,Z 176,A 30.0218,B 6.9591,C 0.1899,E1 7.1026,E2 422.1391} C_DIS
LIN {X 120.1917,Y 72.133,Z 176,A 32.8597,B 6.9593,C 0.1846,E1 7.0986,E2 419.3136} C_DIS
LIN {X 118.1457,Y 75.4364,Z 176,A 34.4785,B 6.9593,C 0.1802,E1 7.0962,E2 417.6901} C_DIS
LIN {X 115.6279,Y 79.2416,Z 176,A 36.2957,B 6.9595,C 0.1766,E1 7.0934,E2 415.8783} C_DIS
LIN {X 113.2022,Y 82.6707,Z 176,A 38.0357,B 6.9595,C 0.1722,E1 7.0906,E2 414.1347} C_DIS
LIN {X 109.9413,Y 86.9589,Z 176,A 40.4652,B 6.9598,C 0.1631,E1 7.0863,E2 411.6749} C_DIS
LIN {X 107.5179,Y 89.9387,Z 176,A 41.6858,B 6.9598,C 0.166,E1 7.0842,E2 410.4988} C_DIS
LIN {X 104.71,Y 93.1936,Z 176,A 43.4405,B 6.9598,C 0.1622,E1 7.081,E2 408.7439} C_DIS
LIN {X 101.8657,Y 96.2935,Z 176,A 45.1337,B 6.9599,C 0.1591,E1 7.0778,E2 407.0536} C_DIS
LIN {X 98.7935,Y 99.4428,Z 176,A 47.0912,B 6.96,C 0.1526,E1 7.0739,E2 405.0751} C_DIS
LIN {X 93.7373,Y 104.2231,Z 176,A 49.4375,B 6.96,C 0.1559,E1 7.0692,E2 402.792} C_DIS
LIN {X 91.213,Y 106.4394,Z 176,A 51.1117,B 6.9601,C 0.148,E1 7.0656,E2 401.079} C_DIS
LIN {X 87.821,Y 109.2546,Z 176,A 52.8408,B 6.9601,C 0.146,E1 7.0619,E2 399.3589} C_DIS
LIN {X 84.3341,Y 111.9679,Z 176,A 54.6291,B 6.9602,C 0.1432,E1 7.0579,E2 397.5726} C_DIS
LIN {X 80.758,Y 114.574,Z 176,A 56.7129,B 6.9604,C 0.1354,E1 7.0531,E2 395.4532} C_DIS
LIN {X 77.6191,Y 116.7235,Z 176,A 57.6538,B 6.9602,C 0.1435,E1 7.0511,E2 394.5907} C_DIS
LIN {X 73.5344,Y 119.339,Z 176,A 59.9087,B 6.9604,C 0.1358,E1 7.0457,E2 392.301} C_DIS
LIN {X 70.3284,Y 121.2558,Z 176,A 61.4493,B 6.9604,C 0.1333,E1 7.042,E2 390.7587} C_DIS
LIN {X 66.33,Y 123.4884,Z 176,A 63.4371,B 6.9605,C 0.1288,E1 7.0371,E2 388.756} C_DIS
LIN {X 59.7525,Y 126.8017,Z 176,A 66.1823,B 6.9605,C 0.1295,E1 7.0303,E2 386.0448} C_DIS
LIN {X 56.4757,Y 128.2952,Z 176,A 68.0153,B 6.9607,C 0.1217,E1 7.0255,E2 384.1659} C_DIS
LIN {X 53.0525,Y 129.7475,Z 176,A 69.0964,B 6.9606,C 0.1273,E1 7.0229,E2 383.1409} C_DIS
LIN {X 50.4935,Y 130.7632,Z 176,A 70.2979,B 6.9606,C 0.1249,E1 7.0197,E2 381.9298} C_DIS
LIN {X 47.1631,Y 132.0012,Z 176,A 71.7264,B 6.9606,C 0.1238,E1 7.016,E2 380.5045} C_DIS
LIN {X 43.9621,Y 133.1013,Z 176,A 73.0856,B 6.9606,C 0.123,E1 7.0124,E2 379.1486} C_DIS
LIN {X 40.2177,Y 134.2824,Z 176,A 74.8406,B 6.9606,C 0.1192,E1 7.0076,E2 377.375} C_DIS
LIN {X 36.1664,Y 135.4272,Z 176,A 76.7348,B 6.9608,C 0.115,E1 7.0025,E2 375.4589} C_DIS
LIN {X 32.6537,Y 136.317,Z 176,A 77.8467,B 6.9607,C 0.12,E1 6.9996,E2 374.3943} C_DIS
LIN {X 29.4371,Y 137.0475,Z 176,A 79.3666,B 6.9607,C 0.1164,E1 6.9954,E2 372.853} C_DIS
LIN {X 26.0077,Y 137.7398,Z 176,A 80.6641,B 6.9607,C 0.1177,E1 6.9919,E2 371.5728} C_DIS
LIN {X 22.5593,Y 138.3471,Z 176,A 82.3927,B 6.9608,C 0.1123,E1 6.987,E2 369.8068} C_DIS
LIN {X 19.0097,Y 138.8797,Z 176,A 83.6651,B 6.9608,C 0.1148,E1 6.9835,E2 368.5598} C_DIS
LIN {X 15.4587,Y 139.3192,Z 176,A 85.0681,B 6.9608,C 0.1153,E1 6.9797,E2 367.1648} C_DIS
LIN {X 11.1121,Y 139.7341,Z 176,A 86.947,B 6.9608,C 0.1133,E1 6.9744,E2 365.2747} C_DIS
LIN {X 6.6307,Y 140.0172,Z 176,A 88.5886,B 6.9608,C 0.116,E1 6.9699,E2 363.6584} C_DIS
LIN {X 2.345,Y 140.154,Z 176,A 90.3513,B 6.9608,C 0.1157,E1 6.965,E2 361.8951} C_DIS
LIN {X -1.5703,Y 140.1669,Z 176,A 92.0938,B 6.9608,C 0.1136,E1 6.9601,E2 360.1353} C_DIS
LIN {X -5.8387,Y 140.0524,Z 176,A 93.933,B 6.9608,C 0.1123,E1 6.9549,E2 358.285} C_DIS
LIN {X -10.6728,Y 139.7674,Z 176,A 96.0054,B 6.9608,C 0.1112,E1 6.9491,E2 356.2018} C_DIS
LIN {X -14.2692,Y 139.4472,Z 176,A 97.2208,B 6.9608,C 0.1156,E1 6.9458,E2 355.0203} C_DIS
LIN {X -18.017,Y 139.0108,Z 176,A 98.7156,B 6.9608,C 0.1168,E1 6.9417,E2 353.5323} C_DIS
LIN {X -24.3437,Y 138.0438,Z 176,A 101.3086,B 6.9608,C 0.1184,E1 6.9346,E2 350.9438} C_DIS
LIN {X -28.4766,Y 137.2513,Z 176,A 102.9958,B 6.9607,C 0.1198,E1 6.9299,E2 349.2618} C_DIS
LIN {X -31.4785,Y 136.5933,Z 176,A 104.3454,B 6.9607,C 0.1192,E1 6.9262,E2 347.9012} C_DIS
LIN {X -35.4487,Y 135.6179,Z 176,A 105.9081,B 6.9607,C 0.1219,E1 6.922,E2 346.3532} C_DIS
LIN {X -38.5739,Y 134.7638,Z 176,A 107.3212,B 6.9607,C 0.1217,E1 6.9182,E2 344.9298} C_DIS
LIN {X -41.2337,Y 133.9714,Z 176,A 108.4947,B 6.9607,C 0.122,E1 6.9151,E2 343.7521} C_DIS
LIN {X -44.9925,Y 132.7582,Z 176,A 110.6661,B 6.9607,C 0.1155,E1 6.9091,E2 341.5111} C_DIS
LIN {X -49.4688,Y 131.1543,Z 176,A 111.9576,B 6.9606,C 0.1267,E1 6.906,E2 340.3037} C_DIS
LIN {X -54.4785,Y 129.1543,Z 176,A 114.286,B 6.9606,C 0.1274,E1 6.8999,E2 337.9614} C_DIS
LIN {X -61.4954,Y 125.9647,Z 176,A 117.3496,B 6.9605,C 0.1324,E1 6.8922,E2 334.9114} C_DIS
LIN {X -63.9378,Y 124.742,Z 176,A 118.6243,B 6.9605,C 0.1316,E1 6.8889,E2 333.6175} C_DIS
LIN {X -67.8055,Y 122.6844,Z 176,A 120.8441,B 6.9605,C 0.1281,E1 6.8834,E2 331.3446} C_DIS
LIN {X -71.4724,Y 120.5855,Z 176,A 122.1307,B 6.9604,C 0.1367,E1 6.8804,E2 330.1154} C_DIS
LIN {X -74.9506,Y 118.4545,Z 176,A 124.0049,B 6.9604,C 0.1364,E1 6.8759,E2 328.2164} C_DIS
LIN {X -79.1032,Y 115.7229,Z 176,A 125.9993,B 6.9604,C 0.1402,E1 6.8713,E2 326.2284} C_DIS
LIN {X -82.9729,Y 112.9802,Z 176,A 128.1963,B 6.9604,C 0.1399,E1 6.8663,E2 324.0002} C_DIS
LIN {X -85.8628,Y 110.7993,Z 176,A 129.7591,B 6.9603,C 0.1414,E1 6.8628,E2 322.4281} C_DIS
LIN {X -89.0596,Y 108.248,Z 176,A 131.1418,B 6.9601,C 0.1483,E1 6.8599,E2 321.0837} C_DIS
LIN {X -95.1448,Y 102.94,Z 176,A 135.2294,B 6.9602,C 0.1441,E1 6.8512,E2 316.8984} C_DIS
LIN {X -99.6934,Y 98.5413,Z 176,A 136.8771,B 6.9598,C 0.1619,E1 6.8482,E2 315.3731} C_DIS
LIN {X -104.7258,Y 93.1758,Z 176,A 140.5935,B 6.9599,C 0.1589,E1 6.841,E2 311.5692} C_DIS
LIN {X -107.7246,Y 89.6916,Z 176,A 141.9769,B 6.9597,C 0.1696,E1 6.8386,E2 310.2508} C_DIS
LIN {X -110.2711,Y 86.5408,Z 176,A 143.8135,B 6.9597,C 0.1709,E1 6.8354,E2 308.3927} C_DIS
LIN {X -112.6239,Y 83.4565,Z 176,A 145.2631,B 6.9595,C 0.1764,E1 6.833,E2 306.962} C_DIS
LIN {X -114.9242,Y 80.2591,Z 176,A 147.0125,B 6.9595,C 0.1784,E1 6.8302,E2 305.1963} C_DIS
LIN {X -117.4639,Y 76.4938,Z 176,A 149.5138,B 6.9595,C 0.1745,E1 6.8262,E2 302.6141} C_DIS
LIN {X -120.4273,Y 71.7378,Z 176,A 151.011,B 6.9591,C 0.1904,E1 6.8242,E2 301.2208} C_DIS
LIN {X -122.7725,Y 67.6465,Z 176,A 153.0025,B 6.9591,C 0.1944,E1 6.8215,E2 299.223} C_DIS
LIN {X -124.3777,Y 64.6452,Z 176,A 154.5834,B 6.959,C 0.1955,E1 6.8194,E2 297.6191} C_DIS
LIN {X -126.5799,Y 60.2168,Z 176,A 156.8983,B 6.959,C 0.197,E1 6.8165,E2 295.2686} C_DIS
LIN {X -128.0409,Y 57.0443,Z 176,A 158.0644,B 6.9587,C 0.2041,E1 6.8152,E2 294.1374} C_DIS
LIN {X -129.5355,Y 53.5658,Z 176,A 159.5917,B 6.9587,C 0.2085,E1 6.8135,E2 292.6141} C_DIS
LIN {X -130.7386,Y 50.5567,Z 176,A 160.9551,B 6.9585,C 0.2115,E1 6.8122,E2 291.247} C_DIS
LIN {X -131.9704,Y 47.2483,Z 176,A 162.4354,B 6.9585,C 0.215,E1 6.8107,E2 289.7633} C_DIS
LIN {X -133.1016,Y 43.9614,Z 176,A 163.951,B 6.9583,C 0.2176,E1 6.8094,E2 288.2369} C_DIS
LIN {X -134.4772,Y 39.5531,Z 176,A 165.8244,B 6.9582,C 0.223,E1 6.8079,E2 286.3671} C_DIS
LIN {X -135.5361,Y 35.7581,Z 176,A 167.428,B 6.958,C 0.2276,E1 6.8067,E2 284.7659} C_DIS
LIN {X -136.3955,Y 32.3278,Z 176,A 168.9173,B 6.9579,C 0.2311,E1 6.8057,E2 283.2723} C_DIS
LIN {X -137.0409,Y 29.4679,Z 176,A 170.2075,B 6.9579,C 0.2333,E1 6.8049,E2 281.9714} C_DIS
LIN {X -138.1664,Y 23.6421,Z 176,A 172.5207,B 6.9575,C 0.2416,E1 6.8038,E2 279.6748} C_DIS
LIN {X -138.786,Y 19.6736,Z 176,A 173.9243,B 6.9573,C 0.2492,E1 6.8032,E2 278.3032} C_DIS
LIN {X -139.1473,Y 16.9336,Z 176,A 176.3017,B 6.9577,C 0.2368,E1 6.8023,E2 275.7659} C_DIS
LIN {X -139.7687,Y 10.6548,Z 176,A 177.9379,B 6.957,C 0.2561,E1 6.802,E2 274.2541} C_DIS
LIN {X -140.1282,Y 3.5808,Z 176,A -179.3877,B 6.9566,C 0.2671,E1 6.8016,E2 271.6107} C_DIS
LIN {X -140.1248,Y -3.7014,Z 176,A -175.7151,B 6.9566,C 0.2671,E1 6.8016,E2 267.8513} C_DIS
LIN {X -139.8305,Y -9.8088,Z 176,A -173.5297,B 6.9562,C 0.2781,E1 6.802,E2 265.7085} C_DIS
LIN {X -139.1825,Y -16.6382,Z 176,A -170.1145,B 6.9562,C 0.2784,E1 6.803,E2 262.2166} C_DIS
LIN {X -138.67,Y -20.4853,Z 176,A -168.9084,B 6.9558,C 0.2877,E1 6.8034,E2 261.0611} C_DIS
LIN {X -138.1347,Y -23.8323,Z 176,A -167.2945,B 6.9558,C 0.2888,E1 6.8042,E2 259.4187} C_DIS
LIN {X -137.3842,Y -27.8235,Z 176,A -165.7003,B 6.9555,C 0.2942,E1 6.805,E2 257.8341} C_DIS
LIN {X -136.5498,Y -31.6691,Z 176,A -164.1458,B 6.9553,C 0.2994,E1 6.806,E2 256.2879} C_DIS
LIN {X -135.8098,Y -34.7029,Z 176,A -162.8366,B 6.9552,C 0.3025,E1 6.8069,E2 254.9753} C_DIS
LIN {X -134.9576,Y -37.8812,Z 176,A -161.4843,B 6.955,C 0.3061,E1 6.8079,E2 253.623} C_DIS
LIN {X -134.0378,Y -41.0169,Z 176,A -160.0619,B 6.955,C 0.3086,E1 6.809,E2 252.1901} C_DIS
LIN {X -132.8469,Y -44.7261,Z 176,A -158.5227,B 6.9547,C 0.3136,E1 6.8103,E2 250.6589} C_DIS
LIN {X -131.3579,Y -48.925,Z 176,A -156.8245,B 6.9544,C 0.3201,E1 6.8119,E2 248.9779} C_DIS
LIN {X -130.2208,Y -51.8782,Z 176,A -155.0949,B 6.9544,C 0.3179,E1 6.8138,E2 247.1923} C_DIS
LIN {X -128.5652,Y -55.8527,Z 176,A -153.4774,B 6.9542,C 0.3243,E1 6.8155,E2 245.5944} C_DIS
LIN {X -126.9929,Y -59.3431,Z 176,A -151.8956,B 6.954,C 0.3281,E1 6.8173,E2 244.0114} C_DIS
LIN {X -125.2698,Y -62.9011,Z 176,A -150.1312,B 6.954,C 0.3303,E1 6.8196,E2 242.2285} C_DIS
LIN {X -120.8981,Y -70.9415,Z 176,A -146.2582,B 6.9536,C 0.3378,E1 6.8248,E2 238.3402} C_DIS
LIN {X -118.2908,Y -75.2096,Z 176,A -144.2949,B 6.9533,C 0.3438,E1 6.8277,E2 236.3886} C_DIS
LIN {X -116.1468,Y -78.4792,Z 176,A -142.6349,B 6.9531,C 0.3467,E1 6.8303,E2 234.7212} C_DIS
LIN {X -113.5356,Y -82.2113,Z 176,A -140.7253,B 6.9529,C 0.3503,E1 6.8334,E2 232.8061} C_DIS
LIN {X -110.7491,Y -85.9283,Z 176,A -138.811,B 6.9527,C 0.3543,E1 6.8366,E2 230.8904} C_DIS
LIN {X -107.8049,Y -89.5946,Z 176,A -136.861,B 6.9525,C 0.3581,E1 6.8401,E2 228.9375} C_DIS
LIN {X -104.8806,Y -93.0007,Z 176,A -135.0257,B 6.9523,C 0.3619,E1 6.8435,E2 227.1028} C_DIS
LIN {X -102.0004,Y -96.1507,Z 176,A -133.2454,B 6.9522,C 0.365,E1 6.8469,E2 225.3183} C_DIS
LIN {X -99.022,Y -99.2158,Z 176,A -131.4547,B 6.952,C 0.3678,E1 6.8504,E2 223.5223} C_DIS
LIN {X -95.8118,Y -102.3196,Z 176,A -129.5641,B 6.952,C 0.3704,E1 6.8542,E2 221.6236} C_DIS
LIN {X -92.4471,Y -105.3694,Z 176,A -127.6911,B 6.9517,C 0.3736,E1 6.8581,E2 219.7487} C_DIS
LIN {X -88.9665,Y -108.3242,Z 176,A -125.8036,B 6.9516,C 0.3765,E1 6.8622,E2 217.8587} C_DIS
LIN {X -85.4767,Y -111.0988,Z 176,A -123.9441,B 6.9514,C 0.3791,E1 6.8663,E2 215.9946} C_DIS
LIN {X -79.6121,Y -115.3736,Z 176,A -121.194,B 6.951,C 0.3869,E1 6.8725,E2 213.2735} C_DIS
LIN {X -76.8833,Y -117.2095,Z 176,A -119.4981,B 6.9512,C 0.3838,E1 6.8765,E2 211.5312} C_DIS
LIN {X -72.5741,Y -119.9252,Z 176,A -117.5282,B 6.9509,C 0.3884,E1 6.8812,E2 209.5763} C_DIS
LIN {X -68.5746,Y -122.2562,Z 176,A -114.4907,B 6.9517,C 0.374,E1 6.889,E2 206.3857} C_DIS
LIN {X -61.1512,Y -126.1335,Z 176,A -112.2678,B 6.9505,C 0.3959,E1 6.8941,E2 204.3234} C_DIS
LIN {X -56.0286,Y -128.4892,Z 176,A -110.0789,B 6.9503,C 0.4001,E1 6.8996,E2 202.1496} C_DIS
LIN {X -53.2294,Y -129.6759,Z 176,A -108.5035,B 6.9505,C 0.3964,E1 6.9038,E2 200.53} C_DIS
LIN {X -49.3022,Y -131.2167,Z 176,A -106.8501,B 6.9503,C 0.399,E1 6.9081,E2 198.8858} C_DIS
LIN {X -45.5084,Y -132.5808,Z 176,A -105.2528,B 6.9503,C 0.4012,E1 6.9123,E2 197.295} C_DIS
LIN {X -41.1419,Y -133.9996,Z 176,A -103.3525,B 6.9501,C 0.4022,E1 6.9174,E2 195.3912} C_DIS
LIN {X -34.3298,Y -135.9045,Z 176,A -100.8549,B 6.9497,C 0.4101,E1 6.924,E2 192.9452} C_DIS
LIN {X -29.7042,Y -136.9899,Z 176,A -98.8023,B 6.9497,C 0.4095,E1 6.9296,E2 190.8776} C_DIS
LIN {X -27.1492,Y -137.5214,Z 176,A -97.4638,B 6.9499,C 0.4058,E1 6.9333,E2 189.5029} C_DIS
LIN {X -22.1783,Y -138.4097,Z 176,A -95.276,B 6.95,C 0.4046,E1 6.9394,E2 187.2979} C_DIS
LIN {X -18.1986,Y -138.987,Z 176,A -93.6885,B 6.95,C 0.4059,E1 6.9438,E2 185.7173} C_DIS
LIN {X -14.819,Y -139.3881,Z 176,A -92.2484,B 6.95,C 0.4054,E1 6.9478,E2 184.2702} C_DIS
LIN {X -10.5006,Y -139.78,Z 176,A -90.5486,B 6.9499,C 0.4068,E1 6.9525,E2 182.5794} C_DIS
LIN {X -7.0233,Y -139.9975,Z 176,A -89.1415,B 6.9499,C 0.4071,E1 6.9564,E2 181.1738} C_DIS
LIN {X -3.0001,Y -140.1431,Z 176,A -87.4117,B 6.9499,C 0.4057,E1 6.9613,E2 179.4322} C_DIS
LIN {X 1.0394,Y -140.169,Z 176,A -85.9235,B 6.9498,C 0.4081,E1 6.9654,E2 177.9649} C_DIS
Enddeposition()
LIN {X 1.0394,Y -140.169,Z 176,A -85.9235,B 6.9498,C 0.4081,E1 6.9654,E2 177.9649} C_DIS
Startdeposition()
$VEL.CP = VEL_PRINT
LIN {X -0.3099,Y -141.0798,Z 176,A -86.9011,B 6.9493,C 0.4192,E1 6.9626,E2 179.0328} C_DIS
LIN {X -3.7372,Y -141.0299,Z 176,A -88.1541,B 6.9494,C 0.417,E1 6.9591,E2 180.268} C_DIS
LIN {X -6.0661,Y -140.9499,Z 176,A -89.3111,B 6.9492,C 0.4204,E1 6.9558,E2 181.4533} C_DIS
LIN {X -9.8463,Y -140.7358,Z 176,A -90.7785,B 6.9492,C 0.4192,E1 6.9517,E2 182.9121} C_DIS
LIN {X -12.6039,Y -140.517,Z 176,A -91.9828,B 6.9492,C 0.4203,E1 6.9483,E2 184.1277} C_DIS
LIN {X -15.6221,Y -140.2126,Z 176,A -93.376,B 6.9491,C 0.4227,E1 6.9444,E2 185.5426} C_DIS
LIN {X -19.9036,Y -139.668,Z 176,A -94.9448,B 6.9493,C 0.4193,E1 6.9401,E2 187.0876} C_DIS
LIN {X -22.9252,Y -139.2043,Z 176,A -96.3782,B 6.9491,C 0.4219,E1 6.9361,E2 188.5468} C_DIS
LIN {X -27.4243,Y -138.3897,Z 176,A -98.0494,B 6.9494,C 0.4182,E1 6.9316,E2 190.1941} C_DIS
LIN {X -31.228,Y -137.5795,Z 176,A -99.7731,B 6.9493,C 0.4197,E1 6.9268,E2 191.9372} C_DIS
LIN {X -35.7613,Y -136.4726,Z 176,A -101.5767,B 6.9494,C 0.4172,E1 6.922,E2 193.7293} C_DIS
LIN {X -40.5376,Y -135.1317,Z 176,A -103.605,B 6.9494,C 0.416,E1 6.9165,E2 195.7599} C_DIS
LIN {X -43.5241,Y -134.1987,Z 176,A -104.8842,B 6.9495,C 0.4152,E1 6.9131,E2 197.0404} C_DIS
LIN {X -47.4082,Y -132.8756,Z 176,A -106.5756,B 6.9495,C 0.4142,E1 6.9086,E2 198.7353} C_DIS
LIN {X -50.7423,Y -131.6382,Z 176,A -108.0522,B 6.9496,C 0.4133,E1 6.9048,E2 200.2164} C_DIS
LIN {X -54.1276,Y -130.2823,Z 176,A -109.5214,B 6.9497,C 0.4117,E1 6.901,E2 201.6841} C_DIS
LIN {X -56.784,Y -129.1493,Z 176,A -110.8598,B 6.9497,C 0.413,E1 6.8975,E2 203.0446} C_DIS
LIN {X -60.6647,Y -127.3696,Z 176,A -112.3775,B 6.95,C 0.4078,E1 6.8937,E2 204.5339} C_DIS
LIN {X -63.8601,Y -125.7979,Z 176,A -113.9028,B 6.95,C 0.4073,E1 6.8899,E2 206.0697} C_DIS
LIN {X -69.4809,Y -122.7858,Z 176,A -116.6414,B 6.95,C 0.4062,E1 6.8831,E2 208.828} C_DIS
LIN {X -73.5291,Y -120.4048,Z 176,A -118.4012,B 6.9503,C 0.4014,E1 6.879,E2 210.5683} C_DIS
LIN {X -76.7631,Y -118.3689,Z 176,A -120.1188,B 6.9503,C 0.4015,E1 6.8749,E2 212.3076} C_DIS
LIN {X -80.7681,Y -115.6735,Z 176,A -121.8947,B 6.9507,C 0.3959,E1 6.8708,E2 214.059} C_DIS
LIN {X -83.8824,Y -113.4359,Z 176,A -123.6768,B 6.9507,C 0.3966,E1 6.8667,E2 215.8705} C_DIS
LIN {X -87.47,Y -110.693,Z 176,A -125.5397,B 6.9507,C 0.3939,E1 6.8626,E2 217.7369} C_DIS
LIN {X -91.0381,Y -107.7777,Z 176,A -127.4675,B 6.9509,C 0.3914,E1 6.8585,E2 219.6717} C_DIS
LIN {X -94.4137,Y -104.8331,Z 176,A -129.2666,B 6.9511,C 0.3878,E1 6.8547,E2 221.4679} C_DIS
LIN {X -97.726,Y -101.7522,Z 176,A -131.0939,B 6.9513,C 0.3842,E1 6.851,E2 223.2934} C_DIS
LIN {X -100.7307,Y -98.778,Z 176,A -132.8248,B 6.9515,C 0.3811,E1 6.8476,E2 225.0256} C_DIS
LIN {X -103.5873,Y -95.7789,Z 176,A -134.5747,B 6.9516,C 0.3786,E1 6.8442,E2 226.7839} C_DIS
Enddeposition()
END
